LIN {X 0,Y 234.876,Z 433.115,A -85,B 0,C 180,E1 -19741.921,E2 -19741.921} C_VEL
LIN {X 0,Y 235.179,Z 429.868,A -85,B 0,C 180,E1 -19746.209,E2 -19746.209} C_VEL
LIN {X 0,Y 235.105,Z 427.906,A -85,B 0,C 180,E1 -19748.993,E2 -19748.993} C_VEL
LIN {X 0,Y 234.901,Z 426.222,A -85,B 0,C 180,E1 -19751.584,E2 -19751.584} C_VEL
LIN {X 0,Y 234.9,Z 426.223,A -85,B 0,C 180,E1 -19755.895,E2 -19755.895} C_VEL
LIN {X 0,Y 234.9,Z 426.226,A -85,B 0,C 180,E1 -19758.835,E2 -19758.835} C_VEL
LIN {X 0,Y 234.957,Z 426.217,A -85,B 0,C 180,E1 -19761.086,E2 -19761.086} C_VEL
LIN {X 0,Y 234.963,Z 426.216,A -85,B 0,C 180,E1 -19765.367,E2 -19765.367} C_VEL
LIN {X 0,Y 234.926,Z 426.22,A -85,B 0,C 180,E1 -19769.431,E2 -19769.431} C_VEL
LIN {X 0,Y 234.996,Z 426.211,A -85,B 0,C 180,E1 -19773.794,E2 -19773.794} C_VEL
LIN {X 0,Y 235.015,Z 426.21,A -85,B 0,C 180,E1 -19778.97,E2 -19778.97} C_VEL
LIN {X 0,Y 235.099,Z 426.198,A -85,B 0,C 180,E1 -19783.059,E2 -19783.059} C_VEL
LIN {X 0,Y 235.15,Z 426.194,A -85,B 0,C 180,E1 -19787.924,E2 -19787.924} C_VEL
LIN {X 0,Y 235.393,Z 426.161,A -85,B 0,C 180,E1 -19791.415,E2 -19791.415} C_VEL
LIN {X 0,Y 235.409,Z 426.16,A -85,B 0,C 180,E1 -19793.141,E2 -19793.141} C_VEL
LIN {X 0,Y 235.598,Z 426.138,A -85,B 0,C 180,E1 -19798.29,E2 -19798.29} C_VEL
LIN {X 0,Y 235.599,Z 426.139,A -85,B 0,C 180,E1 -19801.709,E2 -19801.709} C_VEL
LIN {X 0,Y 235.409,Z 426.161,A -85,B 0,C 180,E1 -19806.858,E2 -19806.858} C_VEL
LIN {X 0,Y 235.256,Z 426.178,A -85,B 0,C 180,E1 -19810.326,E2 -19810.326} C_VEL
LIN {X 0,Y 235.117,Z 426.198,A -85,B 0,C 180,E1 -19815.606,E2 -19815.606} C_VEL
LIN {X 0,Y 235.012,Z 426.212,A -85,B 0,C 180,E1 -19819.205,E2 -19819.205} C_VEL
LIN {X 0,Y 234.964,Z 426.216,A -85,B 0,C 180,E1 -19822.883,E2 -19822.883} C_VEL
LIN {X 0,Y 234.97,Z 426.215,A -85,B 0,C 180,E1 -19826.657,E2 -19826.657} C_VEL
LIN {X 0,Y 234.924,Z 426.222,A -85,B 0,C 180,E1 -19830.569,E2 -19830.569} C_VEL
LIN {X 0,Y 234.929,Z 426.22,A -85,B 0,C 180,E1 -19834.638,E2 -19834.638} C_VEL
LIN {X 0,Y 234.966,Z 426.376,A -85,B 0,C 180,E1 -19838.637,E2 -19838.637} C_VEL
LIN {X 0,Y 235.348,Z 428.729,A -85,B 0,C 180,E1 -19841.707,E2 -19841.707} C_VEL
LIN {X 0,Y 235.874,Z 431.984,A -85,B 0,C 180,E1 -19845.651,E2 -19845.651} C_VEL
LIN {X 0,Y 236.373,Z 435.044,A -85,B 0,C 180,E1 -19849.147,E2 -19849.147} C_VEL
LIN {X 0,Y 236.611,Z 436.635,A -85,B 0,C 180,E1 -19850.894,E2 -19850.894} C_VEL
LIN {X 0,Y 235.984,Z 437.599,A -85,B 0,C 180,E1 -19851.808,E2 -19851.808} C_VEL
LIN {X 0,Y 233.134,Z 439.375,A -85,B 0,C 180,E1 -19853.223,E2 -19853.223} C_VEL
LIN {X 0,Y 230.123,Z 441.18,A -85,B 0,C 180,E1 -19854.668,E2 -19854.668} C_VEL
LIN {X 0,Y 229.299,Z 442.206,A -85,B 0,C 180,E1 -19855.619,E2 -19855.619} C_VEL
LIN {X 0,Y 228.924,Z 443.785,A -85,B 0,C 180,E1 -19857.192,E2 -19857.192} C_VEL
LIN {X 0,Y 229.837,Z 447.058,A -85,B 0,C 180,E1 -19857.512,E2 -19857.512} C_VEL
LIN {X 0,Y 233.319,Z 459.076,A -85,B 0,C 180,E1 -19858.865,E2 -19858.865} C_VEL
LIN {X 0,Y 235.842,Z 471.592,A -85,B 0,C 180,E1 -19860.433,E2 -19860.433} C_VEL
LIN {X 0,Y 237.294,Z 482.933,A -85,B 0,C 180,E1 -19862.06,E2 -19862.06} C_VEL
LIN {X 0,Y 237.835,Z 494.199,A -85,B 0,C 180,E1 -19863.924,E2 -19863.924} C_VEL
LIN {X 0,Y 237.645,Z 500.432,A -85,B 0,C 180,E1 -19865.075,E2 -19865.075} C_VEL
LIN {X 0,Y 235.035,Z 510.888,A -85,B 0,C 180,E1 -19867.125,E2 -19867.125} C_VEL
LIN {X 0,Y 232.818,Z 519.781,A -85,B 0,C 180,E1 -19869.356,E2 -19869.356} C_VEL
LIN {X 0,Y 230.662,Z 527.628,A -85,B 0,C 180,E1 -19871.802,E2 -19871.802} C_VEL
LIN {X 0,Y 228.811,Z 534.295,A -85,B 0,C 180,E1 -19874.409,E2 -19874.409} C_VEL
LIN {X 0,Y 227.212,Z 540.397,A -85,B 0,C 180,E1 -19877.495,E2 -19877.495} C_VEL
LIN {X 0,Y 226.338,Z 544.368,A -85,B 0,C 180,E1 -19880.167,E2 -19880.167} C_VEL
LIN {X 0,Y 225.822,Z 547.305,A -85,B 0,C 180,E1 -19882.849,E2 -19882.849} C_VEL
LIN {X 0,Y 225.58,Z 549.275,A -85,B 0,C 180,E1 -19885.539,E2 -19885.539} C_VEL
LIN {X 0,Y 225.644,Z 550.313,A -85,B 0,C 180,E1 -19888.215,E2 -19888.215} C_VEL
LIN {X 0,Y 225.717,Z 550.528,A -85,B 0,C 180,E1 -19890,E2 -19890} C_VEL
LIN {X 0,Y 225.644,Z 550.303,A -85,B 0,C 180,E1 -19891.785,E2 -19891.785} C_VEL
LIN {X 0,Y 225.59,Z 549.231,A -85,B 0,C 180,E1 -19894.494,E2 -19894.494} C_VEL
LIN {X 0,Y 225.822,Z 547.272,A -85,B 0,C 180,E1 -19897.151,E2 -19897.151} C_VEL
LIN {X 0,Y 226.338,Z 544.321,A -85,B 0,C 180,E1 -19899.833,E2 -19899.833} C_VEL
LIN {X 0,Y 227.211,Z 540.331,A -85,B 0,C 180,E1 -19902.505,E2 -19902.505} C_VEL
LIN {X 0,Y 228.811,Z 534.203,A -85,B 0,C 180,E1 -19905.59,E2 -19905.59} C_VEL
LIN {X 0,Y 230.66,Z 527.515,A -85,B 0,C 180,E1 -19908.198,E2 -19908.198} C_VEL
LIN {X 0,Y 232.86,Z 519.542,A -85,B 0,C 180,E1 -19910.671,E2 -19910.671} C_VEL
LIN {X 0,Y 235.031,Z 510.713,A -85,B 0,C 180,E1 -19912.875,E2 -19912.875} C_VEL
LIN {X 0,Y 237.621,Z 500.209,A -85,B 0,C 180,E1 -19914.927,E2 -19914.927} C_VEL
LIN {X 0,Y 237.682,Z 491.057,A -85,B 0,C 180,E1 -19916.586,E2 -19916.586} C_VEL
LIN {X 0,Y 236.988,Z 480.028,A -85,B 0,C 180,E1 -19918.326,E2 -19918.326} C_VEL
LIN {X 0,Y 235.228,Z 468.348,A -85,B 0,C 180,E1 -19919.952,E2 -19919.952} C_VEL
LIN {X 0,Y 232.386,Z 455.412,A -85,B 0,C 180,E1 -19921.511,E2 -19921.511} C_VEL
LIN {X 0,Y 229.009,Z 444.333,A -85,B 0,C 180,E1 -19922.71,E2 -19922.71} C_VEL
LIN {X 0,Y 228.968,Z 443.753,A -85,B 0,C 180,E1 -19922.786,E2 -19922.786} C_VEL
LIN {X 0,Y 229.564,Z 440.977,A -85,B 0,C 180,E1 -19925.569,E2 -19925.569} C_VEL
LIN {X 0,Y 229.614,Z 437.882,A -85,B 0,C 180,E1 -19928.863,E2 -19928.863} C_VEL
LIN {X 0,Y 229.109,Z 434.593,A -85,B 0,C 180,E1 -19932.59,E2 -19932.59} C_VEL
LIN {X 0,Y 228.455,Z 430.668,A -85,B 0,C 180,E1 -19937.407,E2 -19937.407} C_VEL
LIN {X 0,Y 227.928,Z 427.099,A -85,B 0,C 180,E1 -19942.313,E2 -19942.313} C_VEL
LIN {X 0,Y 227.88,Z 427.104,A -85,B 0,C 180,E1 -19946.377,E2 -19946.377} C_VEL
LIN {X 0,Y 227.905,Z 427.099,A -85,B 0,C 180,E1 -19950.436,E2 -19950.436} C_VEL
LIN {X 0,Y 227.929,Z 427.094,A -85,B 0,C 180,E1 -19954.426,E2 -19954.426} C_VEL
LIN {X 0,Y 227.963,Z 427.091,A -85,B 0,C 180,E1 -19958.287,E2 -19958.287} C_VEL
LIN {X 0,Y 228.036,Z 427.082,A -85,B 0,C 180,E1 -19962.826,E2 -19962.826} C_VEL
LIN {X 0,Y 228.096,Z 427.072,A -85,B 0,C 180,E1 -19967.545,E2 -19967.545} C_VEL
LIN {X 0,Y 228.327,Z 427.043,A -85,B 0,C 180,E1 -19971.147,E2 -19971.147} C_VEL
LIN {X 0,Y 228.36,Z 427.036,A -85,B 0,C 180,E1 -19972.929,E2 -19972.929} C_VEL
LIN {X 0,Y 228.556,Z 427.016,A -85,B 0,C 180,E1 -19978.238,E2 -19978.238} C_VEL
LIN {X 0,Y 228.556,Z 427.015,A -85,B 0,C 180,E1 -19981.762,E2 -19981.762} C_VEL
LIN {X 0,Y 228.36,Z 427.038,A -85,B 0,C 180,E1 -19987.071,E2 -19987.071} C_VEL
LIN {X 0,Y 228.173,Z 427.061,A -85,B 0,C 180,E1 -19990.65,E2 -19990.65} C_VEL
LIN {X 0,Y 228.059,Z 427.077,A -85,B 0,C 180,E1 -19996.102,E2 -19996.102} C_VEL
LIN {X 0,Y 227.944,Z 427.087,A -85,B 0,C 180,E1 -19999.825,E2 -19999.825} C_VEL
LIN {X 0,Y 227.915,Z 427.096,A -85,B 0,C 180,E1 -20003.633,E2 -20003.633} C_VEL
LIN {X 0,Y 227.887,Z 427.099,A -85,B 0,C 180,E1 -20007.555,E2 -20007.555} C_VEL
LIN {X 0,Y 227.874,Z 427.101,A -85,B 0,C 180,E1 -20011.622,E2 -20011.622} C_VEL
LIN {X 0,Y 227.901,Z 427.096,A -85,B 0,C 180,E1 -20015.868,E2 -20015.868} C_VEL
LIN {X 0,Y 227.835,Z 427.104,A -85,B 0,C 180,E1 -20020.375,E2 -20020.375} C_VEL
LIN {X 0,Y 227.837,Z 427.106,A -85,B 0,C 180,E1 -20025.192,E2 -20025.192} C_VEL
LIN {X 0,Y 227.821,Z 427.109,A -85,B 0,C 180,E1 -20027.763,E2 -20027.763} C_VEL
LIN {X 0,Y 228.026,Z 428.595,A -85,B 0,C 180,E1 -20030.402,E2 -20030.402} C_VEL
LIN {X 0,Y 228.119,Z 431.17,A -85,B 0,C 180,E1 -20034.172,E2 -20034.172} C_VEL
LIN {X 0,Y 227.972,Z 433.391,A -85,B 0,C 180,E1 -20037.172,E2 -20037.172} C_VEL
LIN {X 0,Y 229.01,Z 436.551,A -85,B 0,C 180,E1 -20037.515,E2 -20037.515} C_VEL
LIN {X 0,Y 233.221,Z 448,A -85,B 0,C 180,E1 -20038.982,E2 -20038.982} C_VEL
LIN {X 0,Y 236.368,Z 459.105,A -85,B 0,C 180,E1 -20040.527,E2 -20040.527} C_VEL
LIN {X 0,Y 238.444,Z 469.825,A -85,B 0,C 180,E1 -20042.158,E2 -20042.158} C_VEL
LIN {X 0,Y 239.727,Z 480.037,A -85,B 0,C 180,E1 -20043.912,E2 -20043.912} C_VEL
LIN {X 0,Y 239.755,Z 482.646,A -85,B 0,C 180,E1 -20044.382,E2 -20044.382} C_VEL
LIN {X 0,Y 237.488,Z 493.091,A -85,B 0,C 180,E1 -20046.222,E2 -20046.222} C_VEL
LIN {X 0,Y 235.441,Z 501.875,A -85,B 0,C 180,E1 -20048.159,E2 -20048.159} C_VEL
LIN {X 0,Y 232.943,Z 510.862,A -85,B 0,C 180,E1 -20050.617,E2 -20050.617} C_VEL
LIN {X 0,Y 230.757,Z 518.268,A -85,B 0,C 180,E1 -20053.182,E2 -20053.182} C_VEL
LIN {X 0,Y 229.037,Z 524.207,A -85,B 0,C 180,E1 -20055.79,E2 -20055.79} C_VEL
LIN {X 0,Y 227.689,Z 528.899,A -85,B 0,C 180,E1 -20058.426,E2 -20058.426} C_VEL
LIN {X 0,Y 226.768,Z 532.486,A -85,B 0,C 180,E1 -20061.086,E2 -20061.086} C_VEL
LIN {X 0,Y 226.108,Z 535.319,A -85,B 0,C 180,E1 -20064.068,E2 -20064.068} C_VEL
LIN {X 0,Y 225.867,Z 536.717,A -85,B 0,C 180,E1 -20066.432,E2 -20066.432} C_VEL
LIN {X 0,Y 225.748,Z 537.552,A -85,B 0,C 180,E1 -20070,E2 -20070} C_VEL
LIN {X 0,Y 225.753,Z 537.359,A -85,B 0,C 180,E1 -20071.784,E2 -20071.784} C_VEL
LIN {X 0,Y 225.866,Z 536.773,A -85,B 0,C 180,E1 -20073.568,E2 -20073.568} C_VEL
LIN {X 0,Y 226.334,Z 534.45,A -85,B 0,C 180,E1 -20077.135,E2 -20077.135} C_VEL
LIN {X 0,Y 227.024,Z 531.583,A -85,B 0,C 180,E1 -20079.803,E2 -20079.803} C_VEL
LIN {X 0,Y 228.079,Z 527.693,A -85,B 0,C 180,E1 -20082.457,E2 -20082.457} C_VEL
LIN {X 0,Y 229.532,Z 522.672,A -85,B 0,C 180,E1 -20085.086,E2 -20085.086} C_VEL
LIN {X 0,Y 231.355,Z 516.347,A -85,B 0,C 180,E1 -20087.685,E2 -20087.685} C_VEL
LIN {X 0,Y 233.68,Z 508.429,A -85,B 0,C 180,E1 -20090.235,E2 -20090.235} C_VEL
LIN {X 0,Y 235.682,Z 500.566,A -85,B 0,C 180,E1 -20092.293,E2 -20092.293} C_VEL
LIN {X 0,Y 238.072,Z 490.511,A -85,B 0,C 180,E1 -20094.412,E2 -20094.412} C_VEL
LIN {X 0,Y 239.88,Z 482.103,A -85,B 0,C 180,E1 -20095.837,E2 -20095.837} C_VEL
LIN {X 0,Y 238.84,Z 471.948,A -85,B 0,C 180,E1 -20097.622,E2 -20097.622} C_VEL
LIN {X 0,Y 236.695,Z 460.288,A -85,B 0,C 180,E1 -20099.439,E2 -20099.439} C_VEL
LIN {X 0,Y 233.574,Z 448.999,A -85,B 0,C 180,E1 -20101.025,E2 -20101.025} C_VEL
LIN {X 0,Y 229.182,Z 436.839,A -85,B 0,C 180,E1 -20102.586,E2 -20102.586} C_VEL
LIN {X 0,Y 227.977,Z 433.327,A -85,B 0,C 180,E1 -20103.023,E2 -20103.023} C_VEL
LIN {X 0,Y 228.157,Z 430.599,A -85,B 0,C 180,E1 -20106.785,E2 -20106.785} C_VEL
LIN {X 0,Y 227.985,Z 428.215,A -85,B 0,C 180,E1 -20110.343,E2 -20110.343} C_VEL
LIN {X 0,Y 227.824,Z 427.103,A -85,B 0,C 180,E1 -20112.238,E2 -20112.238} C_VEL
LIN {X 0,Y 227.838,Z 427.104,A -85,B 0,C 180,E1 -20115.192,E2 -20115.192} C_VEL
LIN {X 0,Y 227.836,Z 427.103,A -85,B 0,C 180,E1 -20119.625,E2 -20119.625} C_VEL
LIN {X 0,Y 227.902,Z 427.095,A -85,B 0,C 180,E1 -20124.132,E2 -20124.132} C_VEL
LIN {X 0,Y 227.872,Z 427.101,A -85,B 0,C 180,E1 -20128.378,E2 -20128.378} C_VEL
LIN {X 0,Y 227.882,Z 427.1,A -85,B 0,C 180,E1 -20132.444,E2 -20132.444} C_VEL
LIN {X 0,Y 227.917,Z 427.096,A -85,B 0,C 180,E1 -20136.368,E2 -20136.368} C_VEL
LIN {X 0,Y 227.946,Z 427.091,A -85,B 0,C 180,E1 -20140.175,E2 -20140.175} C_VEL
LIN {X 0,Y 228.061,Z 427.077,A -85,B 0,C 180,E1 -20143.898,E2 -20143.898} C_VEL
LIN {X 0,Y 228.174,Z 427.062,A -85,B 0,C 180,E1 -20149.35,E2 -20149.35} C_VEL
LIN {X 0,Y 228.361,Z 427.038,A -85,B 0,C 180,E1 -20152.929,E2 -20152.929} C_VEL
LIN {X 0,Y 228.557,Z 427.015,A -85,B 0,C 180,E1 -20158.238,E2 -20158.238} C_VEL
LIN {X 0,Y 228.558,Z 427.016,A -85,B 0,C 180,E1 -20161.762,E2 -20161.762} C_VEL
LIN {X 0,Y 228.361,Z 427.039,A -85,B 0,C 180,E1 -20167.071,E2 -20167.071} C_VEL
LIN {X 0,Y 228.174,Z 427.06,A -85,B 0,C 180,E1 -20170.65,E2 -20170.65} C_VEL
LIN {X 0,Y 228.06,Z 427.077,A -85,B 0,C 180,E1 -20176.102,E2 -20176.102} C_VEL
LIN {X 0,Y 227.945,Z 427.091,A -85,B 0,C 180,E1 -20179.825,E2 -20179.825} C_VEL
LIN {X 0,Y 227.917,Z 427.095,A -85,B 0,C 180,E1 -20183.632,E2 -20183.632} C_VEL
LIN {X 0,Y 227.881,Z 427.098,A -85,B 0,C 180,E1 -20187.556,E2 -20187.556} C_VEL
LIN {X 0,Y 227.869,Z 427.093,A -85,B 0,C 180,E1 -20191.623,E2 -20191.623} C_VEL
LIN {X 0,Y 227.882,Z 427.098,A -85,B 0,C 180,E1 -20195.872,E2 -20195.872} C_VEL
LIN {X 0,Y 227.929,Z 427.222,A -85,B 0,C 180,E1 -20197.88,E2 -20197.88} C_VEL
LIN {X 0,Y 228.462,Z 430.743,A -85,B 0,C 180,E1 -20202.592,E2 -20202.592} C_VEL
LIN {X 0,Y 228.782,Z 432.699,A -85,B 0,C 180,E1 -20205.045,E2 -20205.045} C_VEL
LIN {X 0,Y 229.313,Z 435.857,A -85,B 0,C 180,E1 -20208.782,E2 -20208.782} C_VEL
LIN {X 0,Y 229.629,Z 438.973,A -85,B 0,C 180,E1 -20212.257,E2 -20212.257} C_VEL
LIN {X 0,Y 229.56,Z 441.027,A -85,B 0,C 180,E1 -20214.43,E2 -20214.43} C_VEL
LIN {X 0,Y 229.299,Z 442.206,A -85,B 0,C 180,E1 -20215.619,E2 -20215.619} C_VEL
LIN {X 0,Y 229.36,Z 443.899,A -85,B 0,C 180,E1 -20216.45,E2 -20216.45} C_VEL
LIN {X 0,Y 229.668,Z 446.642,A -85,B 0,C 180,E1 -20217.102,E2 -20217.102} C_VEL
LIN {X 0,Y 230.066,Z 451.856,A -85,B 0,C 180,E1 -20217.799,E2 -20217.799} C_VEL
LIN {X 0,Y 229.581,Z 462.151,A -85,B 0,C 180,E1 -20218.575,E2 -20218.575} C_VEL
LIN {X 0,Y 228.882,Z 468.288,A -85,B 0,C 180,E1 -20219.093,E2 -20219.093} C_VEL
LIN {X 0,Y 228.999,Z 470.221,A -85,B 0,C 180,E1 -20219.327,E2 -20219.327} C_VEL
LIN {X 0,Y 230.592,Z 481.763,A -85,B 0,C 180,E1 -20221.038,E2 -20221.038} C_VEL
LIN {X 0,Y 231.158,Z 492.673,A -85,B 0,C 180,E1 -20222.867,E2 -20222.867} C_VEL
LIN {X 0,Y 230.941,Z 501.408,A -85,B 0,C 180,E1 -20224.542,E2 -20224.542} C_VEL
LIN {X 0,Y 228.484,Z 510.686,A -85,B 0,C 180,E1 -20226.43,E2 -20226.43} C_VEL
LIN {X 0,Y 225.941,Z 520.317,A -85,B 0,C 180,E1 -20228.934,E2 -20228.934} C_VEL
LIN {X 0,Y 223.909,Z 527.425,A -85,B 0,C 180,E1 -20231.233,E2 -20231.233} C_VEL
LIN {X 0,Y 221.938,Z 534.091,A -85,B 0,C 180,E1 -20233.914,E2 -20233.914} C_VEL
LIN {X 0,Y 220.231,Z 540.193,A -85,B 0,C 180,E1 -20237.092,E2 -20237.092} C_VEL
LIN {X 0,Y 219.323,Z 544.164,A -85,B 0,C 180,E1 -20239.849,E2 -20239.849} C_VEL
LIN {X 0,Y 218.76,Z 547.101,A -85,B 0,C 180,E1 -20242.617,E2 -20242.617} C_VEL
LIN {X 0,Y 218.481,Z 549.232,A -85,B 0,C 180,E1 -20245.708,E2 -20245.708} C_VEL
LIN {X 0,Y 218.542,Z 550.109,A -85,B 0,C 180,E1 -20248.157,E2 -20248.157} C_VEL
LIN {X 0,Y 218.631,Z 550.325,A -85,B 0,C 180,E1 -20250,E2 -20250} C_VEL
LIN {X 0,Y 218.542,Z 550.099,A -85,B 0,C 180,E1 -20251.843,E2 -20251.843} C_VEL
LIN {X 0,Y 218.488,Z 549.205,A -85,B 0,C 180,E1 -20254.315,E2 -20254.315} C_VEL
LIN {X 0,Y 218.76,Z 547.067,A -85,B 0,C 180,E1 -20257.383,E2 -20257.383} C_VEL
LIN {X 0,Y 219.323,Z 544.115,A -85,B 0,C 180,E1 -20260.151,E2 -20260.151} C_VEL
LIN {X 0,Y 220.231,Z 540.124,A -85,B 0,C 180,E1 -20262.908,E2 -20262.908} C_VEL
LIN {X 0,Y 221.937,Z 533.996,A -85,B 0,C 180,E1 -20266.086,E2 -20266.086} C_VEL
LIN {X 0,Y 223.907,Z 527.308,A -85,B 0,C 180,E1 -20268.767,E2 -20268.767} C_VEL
LIN {X 0,Y 226.344,Z 518.762,A -85,B 0,C 180,E1 -20271.477,E2 -20271.477} C_VEL
LIN {X 0,Y 228.48,Z 510.505,A -85,B 0,C 180,E1 -20273.57,E2 -20273.57} C_VEL
LIN {X 0,Y 231.06,Z 499.997,A -85,B 0,C 180,E1 -20275.685,E2 -20275.685} C_VEL
LIN {X 0,Y 231.047,Z 489.297,A -85,B 0,C 180,E1 -20277.676,E2 -20277.676} C_VEL
LIN {X 0,Y 230.189,Z 478.595,A -85,B 0,C 180,E1 -20279.412,E2 -20279.412} C_VEL
LIN {X 0,Y 228.305,Z 466.709,A -85,B 0,C 180,E1 -20281.111,E2 -20281.111} C_VEL
LIN {X 0,Y 225.499,Z 454.685,A -85,B 0,C 180,E1 -20282.624,E2 -20282.624} C_VEL
LIN {X 0,Y 222.259,Z 444.269,A -85,B 0,C 180,E1 -20283.826,E2 -20283.826} C_VEL
LIN {X 0,Y 222.193,Z 443.529,A -85,B 0,C 180,E1 -20283.907,E2 -20283.907} C_VEL
LIN {X 0,Y 222.599,Z 439.832,A -85,B 0,C 180,E1 -20287.879,E2 -20287.879} C_VEL
LIN {X 0,Y 222.399,Z 437.38,A -85,B 0,C 180,E1 -20290.675,E2 -20290.675} C_VEL
LIN {X 0,Y 221.861,Z 434.498,A -85,B 0,C 180,E1 -20294.179,E2 -20294.179} C_VEL
LIN {X 0,Y 221.353,Z 431.385,A -85,B 0,C 180,E1 -20298.183,E2 -20298.183} C_VEL
LIN {X 0,Y 220.856,Z 427.981,A -85,B 0,C 180,E1 -20303.013,E2 -20303.013} C_VEL
LIN {X 0,Y 220.817,Z 427.983,A -85,B 0,C 180,E1 -20307.244,E2 -20307.244} C_VEL
LIN {X 0,Y 220.828,Z 427.978,A -85,B 0,C 180,E1 -20311.485,E2 -20311.485} C_VEL
LIN {X 0,Y 220.868,Z 427.972,A -85,B 0,C 180,E1 -20315.565,E2 -20315.565} C_VEL
LIN {X 0,Y 220.894,Z 427.97,A -85,B 0,C 180,E1 -20319.514,E2 -20319.514} C_VEL
LIN {X 0,Y 221.018,Z 427.954,A -85,B 0,C 180,E1 -20323.37,E2 -20323.37} C_VEL
LIN {X 0,Y 221.118,Z 427.941,A -85,B 0,C 180,E1 -20329.006,E2 -20329.006} C_VEL
LIN {X 0,Y 221.313,Z 427.915,A -85,B 0,C 180,E1 -20332.702,E2 -20332.702} C_VEL
LIN {X 0,Y 221.514,Z 427.892,A -85,B 0,C 180,E1 -20338.182,E2 -20338.182} C_VEL
LIN {X 0,Y 221.514,Z 427.893,A -85,B 0,C 180,E1 -20341.818,E2 -20341.818} C_VEL
LIN {X 0,Y 221.313,Z 427.916,A -85,B 0,C 180,E1 -20347.298,E2 -20347.298} C_VEL
LIN {X 0,Y 221.118,Z 427.939,A -85,B 0,C 180,E1 -20350.994,E2 -20350.994} C_VEL
LIN {X 0,Y 221.018,Z 427.953,A -85,B 0,C 180,E1 -20356.63,E2 -20356.63} C_VEL
LIN {X 0,Y 220.894,Z 427.968,A -85,B 0,C 180,E1 -20360.486,E2 -20360.486} C_VEL
LIN {X 0,Y 220.869,Z 427.971,A -85,B 0,C 180,E1 -20364.435,E2 -20364.435} C_VEL
LIN {X 0,Y 220.837,Z 427.975,A -85,B 0,C 180,E1 -20368.514,E2 -20368.514} C_VEL
LIN {X 0,Y 220.826,Z 427.976,A -85,B 0,C 180,E1 -20372.755,E2 -20372.755} C_VEL
LIN {X 0,Y 220.839,Z 427.977,A -85,B 0,C 180,E1 -20377.288,E2 -20377.288} C_VEL
LIN {X 0,Y 220.777,Z 427.985,A -85,B 0,C 180,E1 -20381.951,E2 -20381.951} C_VEL
LIN {X 0,Y 220.777,Z 427.985,A -85,B 0,C 180,E1 -20385.547,E2 -20385.547} C_VEL
LIN {X 0,Y 220.772,Z 427.986,A -85,B 0,C 180,E1 -20387.069,E2 -20387.069} C_VEL
LIN {X 0,Y 221.048,Z 429.859,A -85,B 0,C 180,E1 -20390.515,E2 -20390.515} C_VEL
LIN {X 0,Y 221.109,Z 431.393,A -85,B 0,C 180,E1 -20392.849,E2 -20392.849} C_VEL
LIN {X 0,Y 221.023,Z 433.72,A -85,B 0,C 180,E1 -20396.005,E2 -20396.005} C_VEL
LIN {X 0,Y 222.132,Z 436.853,A -85,B 0,C 180,E1 -20396.382,E2 -20396.382} C_VEL
LIN {X 0,Y 226.152,Z 447.303,A -85,B 0,C 180,E1 -20397.816,E2 -20397.816} C_VEL
LIN {X 0,Y 229.51,Z 458.684,A -85,B 0,C 180,E1 -20399.48,E2 -20399.48} C_VEL
LIN {X 0,Y 231.763,Z 470.005,A -85,B 0,C 180,E1 -20401.276,E2 -20401.276} C_VEL
LIN {X 0,Y 233.049,Z 480.257,A -85,B 0,C 180,E1 -20403.106,E2 -20403.106} C_VEL
LIN {X 0,Y 233.11,Z 484.141,A -85,B 0,C 180,E1 -20403.837,E2 -20403.837} C_VEL
LIN {X 0,Y 230.77,Z 494.355,A -85,B 0,C 180,E1 -20405.725,E2 -20405.725} C_VEL
LIN {X 0,Y 228.452,Z 503.743,A -85,B 0,C 180,E1 -20407.93,E2 -20407.93} C_VEL
LIN {X 0,Y 225.856,Z 512.416,A -85,B 0,C 180,E1 -20410.457,E2 -20410.457} C_VEL
LIN {X 0,Y 223.669,Z 519.583,A -85,B 0,C 180,E1 -20413.103,E2 -20413.103} C_VEL
LIN {X 0,Y 222.162,Z 524.412,A -85,B 0,C 180,E1 -20415.341,E2 -20415.341} C_VEL
LIN {X 0,Y 220.722,Z 529.104,A -85,B 0,C 180,E1 -20418.056,E2 -20418.056} C_VEL
LIN {X 0,Y 219.766,Z 532.69,A -85,B 0,C 180,E1 -20420.799,E2 -20420.799} C_VEL
LIN {X 0,Y 219,Z 535.748,A -85,B 0,C 180,E1 -20424.174,E2 -20424.174} C_VEL
LIN {X 0,Y 218.778,Z 536.921,A -85,B 0,C 180,E1 -20426.317,E2 -20426.317} C_VEL
LIN {X 0,Y 218.674,Z 537.529,A -85,B 0,C 180,E1 -20428.158,E2 -20428.158} C_VEL
LIN {X 0,Y 218.663,Z 537.756,A -85,B 0,C 180,E1 -20430,E2 -20430} C_VEL
LIN {X 0,Y 218.673,Z 537.563,A -85,B 0,C 180,E1 -20431.842,E2 -20431.842} C_VEL
LIN {X 0,Y 218.777,Z 536.977,A -85,B 0,C 180,E1 -20433.684,E2 -20433.684} C_VEL
LIN {X 0,Y 219.045,Z 535.757,A -85,B 0,C 180,E1 -20435.939,E2 -20435.939} C_VEL
LIN {X 0,Y 219.766,Z 532.84,A -85,B 0,C 180,E1 -20439.201,E2 -20439.201} C_VEL
LIN {X 0,Y 220.71,Z 529.31,A -85,B 0,C 180,E1 -20441.946,E2 -20441.946} C_VEL
LIN {X 0,Y 222.12,Z 524.673,A -85,B 0,C 180,E1 -20444.663,E2 -20444.663} C_VEL
LIN {X 0,Y 224.219,Z 517.684,A -85,B 0,C 180,E1 -20447.795,E2 -20447.795} C_VEL
LIN {X 0,Y 226.606,Z 510.101,A -85,B 0,C 180,E1 -20450.421,E2 -20450.421} C_VEL
LIN {X 0,Y 228.958,Z 501.382,A -85,B 0,C 180,E1 -20452.819,E2 -20452.819} C_VEL
LIN {X 0,Y 231.363,Z 491.777,A -85,B 0,C 180,E1 -20454.928,E2 -20454.928} C_VEL
LIN {X 0,Y 233.28,Z 483.589,A -85,B 0,C 180,E1 -20456.383,E2 -20456.383} C_VEL
LIN {X 0,Y 232.443,Z 474.156,A -85,B 0,C 180,E1 -20458.136,E2 -20458.136} C_VEL
LIN {X 0,Y 230.565,Z 463.118,A -85,B 0,C 180,E1 -20459.973,E2 -20459.973} C_VEL
LIN {X 0,Y 228.009,Z 453.076,A -85,B 0,C 180,E1 -20461.498,E2 -20461.498} C_VEL
LIN {X 0,Y 223.602,Z 440.285,A -85,B 0,C 180,E1 -20463.301,E2 -20463.301} C_VEL
LIN {X 0,Y 221.116,Z 434.19,A -85,B 0,C 180,E1 -20464.106,E2 -20464.106} C_VEL
LIN {X 0,Y 221.004,Z 433.54,A -85,B 0,C 180,E1 -20464.227,E2 -20464.227} C_VEL
LIN {X 0,Y 221.141,Z 431.337,A -85,B 0,C 180,E1 -20467.39,E2 -20467.39} C_VEL
LIN {X 0,Y 221.001,Z 429.484,A -85,B 0,C 180,E1 -20470.251,E2 -20470.251} C_VEL
LIN {X 0,Y 220.775,Z 427.981,A -85,B 0,C 180,E1 -20472.931,E2 -20472.931} C_VEL
LIN {X 0,Y 220.773,Z 427.985,A -85,B 0,C 180,E1 -20477.069,E2 -20477.069} C_VEL
LIN {X 0,Y 220.812,Z 427.981,A -85,B 0,C 180,E1 -20480.464,E2 -20480.464} C_VEL
LIN {X 0,Y 220.835,Z 427.978,A -85,B 0,C 180,E1 -20482.795,E2 -20482.795} C_VEL
LIN {X 0,Y 220.826,Z 427.975,A -85,B 0,C 180,E1 -20487.245,E2 -20487.245} C_VEL
LIN {X 0,Y 220.83,Z 427.976,A -85,B 0,C 180,E1 -20491.485,E2 -20491.485} C_VEL
LIN {X 0,Y 220.87,Z 427.97,A -85,B 0,C 180,E1 -20495.565,E2 -20495.565} C_VEL
LIN {X 0,Y 220.896,Z 427.968,A -85,B 0,C 180,E1 -20499.514,E2 -20499.514} C_VEL
LIN {X 0,Y 221.019,Z 427.952,A -85,B 0,C 180,E1 -20503.37,E2 -20503.37} C_VEL
LIN {X 0,Y 221.12,Z 427.94,A -85,B 0,C 180,E1 -20509.006,E2 -20509.006} C_VEL
LIN {X 0,Y 221.314,Z 427.916,A -85,B 0,C 180,E1 -20512.702,E2 -20512.702} C_VEL
LIN {X 0,Y 221.515,Z 427.893,A -85,B 0,C 180,E1 -20518.182,E2 -20518.182} C_VEL
LIN {X 0,Y 221.516,Z 427.892,A -85,B 0,C 180,E1 -20521.818,E2 -20521.818} C_VEL
LIN {X 0,Y 221.314,Z 427.918,A -85,B 0,C 180,E1 -20527.298,E2 -20527.298} C_VEL
LIN {X 0,Y 221.12,Z 427.94,A -85,B 0,C 180,E1 -20530.994,E2 -20530.994} C_VEL
LIN {X 0,Y 221.019,Z 427.953,A -85,B 0,C 180,E1 -20536.63,E2 -20536.63} C_VEL
LIN {X 0,Y 220.895,Z 427.968,A -85,B 0,C 180,E1 -20540.486,E2 -20540.486} C_VEL
LIN {X 0,Y 220.87,Z 427.971,A -85,B 0,C 180,E1 -20544.435,E2 -20544.435} C_VEL
LIN {X 0,Y 220.829,Z 427.973,A -85,B 0,C 180,E1 -20548.515,E2 -20548.515} C_VEL
LIN {X 0,Y 220.818,Z 427.963,A -85,B 0,C 180,E1 -20552.756,E2 -20552.756} C_VEL
LIN {X 0,Y 220.89,Z 428.16,A -85,B 0,C 180,E1 -20557.194,E2 -20557.194} C_VEL
LIN {X 0,Y 221.36,Z 431.471,A -85,B 0,C 180,E1 -20561.815,E2 -20561.815} C_VEL
LIN {X 0,Y 221.862,Z 434.559,A -85,B 0,C 180,E1 -20565.821,E2 -20565.821} C_VEL
LIN {X 0,Y 222.373,Z 437.454,A -85,B 0,C 180,E1 -20569.333,E2 -20569.333} C_VEL
LIN {X 0,Y 222.602,Z 439.883,A -85,B 0,C 180,E1 -20572.12,E2 -20572.12} C_VEL
LIN {X 0,Y 222.544,Z 441.825,A -85,B 0,C 180,E1 -20574.252,E2 -20574.252} C_VEL
LIN {X 0,Y 222.151,Z 443.548,A -85,B 0,C 180,E1 -20576.053,E2 -20576.053} C_VEL
LIN {X 0,Y 223.067,Z 446.896,A -85,B 0,C 180,E1 -20576.401,E2 -20576.401} C_VEL
LIN {X 0,Y 226.804,Z 459.479,A -85,B 0,C 180,E1 -20577.918,E2 -20577.918} C_VEL
LIN {X 0,Y 228.999,Z 470.221,A -85,B 0,C 180,E1 -20579.327,E2 -20579.327} C_VEL
LIN {X 0,Y 229.194,Z 475.519,A -85,B 0,C 180,E1 -20579.991,E2 -20579.991} C_VEL
LIN {X 0,Y 228.397,Z 480.869,A -85,B 0,C 180,E1 -20580.607,E2 -20580.607} C_VEL
LIN {X 0,Y 225.297,Z 492.988,A -85,B 0,C 180,E1 -20582.181,E2 -20582.181} C_VEL
LIN {X 0,Y 224.578,Z 497.835,A -85,B 0,C 180,E1 -20583.053,E2 -20583.053} C_VEL
LIN {X 0,Y 224.246,Z 502.333,A -85,B 0,C 180,E1 -20583.974,E2 -20583.974} C_VEL
LIN {X 0,Y 221.473,Z 512.28,A -85,B 0,C 180,E1 -20586.134,E2 -20586.134} C_VEL
LIN {X 0,Y 219.107,Z 520.782,A -85,B 0,C 180,E1 -20588.465,E2 -20588.465} C_VEL
LIN {X 0,Y 216.784,Z 528.459,A -85,B 0,C 180,E1 -20591.083,E2 -20591.083} C_VEL
LIN {X 0,Y 214.818,Z 534.883,A -85,B 0,C 180,E1 -20593.854,E2 -20593.854} C_VEL
LIN {X 0,Y 213.266,Z 539.988,A -85,B 0,C 180,E1 -20596.663,E2 -20596.663} C_VEL
LIN {X 0,Y 212.309,Z 543.96,A -85,B 0,C 180,E1 -20599.51,E2 -20599.51} C_VEL
LIN {X 0,Y 211.688,Z 546.896,A -85,B 0,C 180,E1 -20602.368,E2 -20602.368} C_VEL
LIN {X 0,Y 211.393,Z 549.152,A -85,B 0,C 180,E1 -20605.855,E2 -20605.855} C_VEL
LIN {X 0,Y 211.442,Z 549.905,A -85,B 0,C 180,E1 -20608.095,E2 -20608.095} C_VEL
LIN {X 0,Y 211.547,Z 550.121,A -85,B 0,C 180,E1 -20610,E2 -20610} C_VEL
LIN {X 0,Y 211.442,Z 549.894,A -85,B 0,C 180,E1 -20611.905,E2 -20611.905} C_VEL
LIN {X 0,Y 211.492,Z 548.271,A -85,B 0,C 180,E1 -20615.721,E2 -20615.721} C_VEL
LIN {X 0,Y 211.688,Z 546.861,A -85,B 0,C 180,E1 -20617.631,E2 -20617.631} C_VEL
LIN {X 0,Y 212.309,Z 543.909,A -85,B 0,C 180,E1 -20620.49,E2 -20620.49} C_VEL
LIN {X 0,Y 213.266,Z 539.917,A -85,B 0,C 180,E1 -20623.337,E2 -20623.337} C_VEL
LIN {X 0,Y 215.101,Z 533.79,A -85,B 0,C 180,E1 -20626.612,E2 -20626.612} C_VEL
LIN {X 0,Y 217.188,Z 527.102,A -85,B 0,C 180,E1 -20629.371,E2 -20629.371} C_VEL
LIN {X 0,Y 219.628,Z 518.869,A -85,B 0,C 180,E1 -20632.065,E2 -20632.065} C_VEL
LIN {X 0,Y 221.987,Z 510.298,A -85,B 0,C 180,E1 -20634.304,E2 -20634.304} C_VEL
LIN {X 0,Y 224.394,Z 500.966,A -85,B 0,C 180,E1 -20636.257,E2 -20636.257} C_VEL
LIN {X 0,Y 224.477,Z 490.217,A -85,B 0,C 180,E1 -20638.358,E2 -20638.358} C_VEL
LIN {X 0,Y 223.708,Z 479.579,A -85,B 0,C 180,E1 -20640.176,E2 -20640.176} C_VEL
LIN {X 0,Y 221.894,Z 467.664,A -85,B 0,C 180,E1 -20641.982,E2 -20641.982} C_VEL
LIN {X 0,Y 219.256,Z 456.069,A -85,B 0,C 180,E1 -20643.55,E2 -20643.55} C_VEL
LIN {X 0,Y 216.024,Z 445.968,A -85,B 0,C 180,E1 -20644.829,E2 -20644.829} C_VEL
LIN {X 0,Y 215.344,Z 443.298,A -85,B 0,C 180,E1 -20645.156,E2 -20645.156} C_VEL
LIN {X 0,Y 215.57,Z 440.315,A -85,B 0,C 180,E1 -20648.515,E2 -20648.515} C_VEL
LIN {X 0,Y 215.292,Z 437.961,A -85,B 0,C 180,E1 -20651.339,E2 -20651.339} C_VEL
LIN {X 0,Y 214.576,Z 433.889,A -85,B 0,C 180,E1 -20656.543,E2 -20656.543} C_VEL
LIN {X 0,Y 214.307,Z 432.098,A -85,B 0,C 180,E1 -20659.013,E2 -20659.013} C_VEL
LIN {X 0,Y 213.8,Z 428.86,A -85,B 0,C 180,E1 -20663.941,E2 -20663.941} C_VEL
LIN {X 0,Y 213.781,Z 428.859,A -85,B 0,C 180,E1 -20668.731,E2 -20668.731} C_VEL
LIN {X 0,Y 213.827,Z 428.851,A -85,B 0,C 180,E1 -20672.603,E2 -20672.603} C_VEL
LIN {X 0,Y 213.853,Z 428.848,A -85,B 0,C 180,E1 -20676.953,E2 -20676.953} C_VEL
LIN {X 0,Y 213.945,Z 428.837,A -85,B 0,C 180,E1 -20682.804,E2 -20682.804} C_VEL
LIN {X 0,Y 213.983,Z 428.832,A -85,B 0,C 180,E1 -20686.708,E2 -20686.708} C_VEL
LIN {X 0,Y 214.198,Z 428.804,A -85,B 0,C 180,E1 -20690.558,E2 -20690.558} C_VEL
LIN {X 0,Y 214.25,Z 428.796,A -85,B 0,C 180,E1 -20692.46,E2 -20692.46} C_VEL
LIN {X 0,Y 214.447,Z 428.772,A -85,B 0,C 180,E1 -20698.122,E2 -20698.122} C_VEL
LIN {X 0,Y 214.556,Z 428.759,A -85,B 0,C 180,E1 -20700,E2 -20700} C_VEL
LIN {X 0,Y 214.447,Z 428.773,A -85,B 0,C 180,E1 -20701.878,E2 -20701.878} C_VEL
LIN {X 0,Y 214.25,Z 428.797,A -85,B 0,C 180,E1 -20707.54,E2 -20707.54} C_VEL
LIN {X 0,Y 214.049,Z 428.82,A -85,B 0,C 180,E1 -20711.362,E2 -20711.362} C_VEL
LIN {X 0,Y 213.936,Z 428.836,A -85,B 0,C 180,E1 -20715.237,E2 -20715.237} C_VEL
LIN {X 0,Y 213.841,Z 428.843,A -85,B 0,C 180,E1 -20719.187,E2 -20719.187} C_VEL
LIN {X 0,Y 213.849,Z 428.846,A -85,B 0,C 180,E1 -20723.227,E2 -20723.227} C_VEL
LIN {X 0,Y 213.83,Z 428.849,A -85,B 0,C 180,E1 -20727.45,E2 -20727.45} C_VEL
LIN {X 0,Y 213.781,Z 428.856,A -85,B 0,C 180,E1 -20731.736,E2 -20731.736} C_VEL
LIN {X 0,Y 213.754,Z 428.858,A -85,B 0,C 180,E1 -20736.287,E2 -20736.287} C_VEL
LIN {X 0,Y 213.719,Z 428.864,A -85,B 0,C 180,E1 -20741.124,E2 -20741.124} C_VEL
LIN {X 0,Y 213.71,Z 428.864,A -85,B 0,C 180,E1 -20743.678,E2 -20743.678} C_VEL
LIN {X 0,Y 213.711,Z 428.867,A -85,B 0,C 180,E1 -20746.343,E2 -20746.343} C_VEL
LIN {X 0,Y 213.932,Z 430.195,A -85,B 0,C 180,E1 -20749.077,E2 -20749.077} C_VEL
LIN {X 0,Y 214.092,Z 431.99,A -85,B 0,C 180,E1 -20751.985,E2 -20751.985} C_VEL
LIN {X 0,Y 214.01,Z 433.796,A -85,B 0,C 180,E1 -20754.709,E2 -20754.709} C_VEL
LIN {X 0,Y 215.21,Z 437.146,A -85,B 0,C 180,E1 -20755.15,E2 -20755.15} C_VEL
LIN {X 0,Y 218.593,Z 445.359,A -85,B 0,C 180,E1 -20756.36,E2 -20756.36} C_VEL
LIN {X 0,Y 222.223,Z 456.62,A -85,B 0,C 180,E1 -20758.09,E2 -20758.09} C_VEL
LIN {X 0,Y 224.486,Z 466.327,A -85,B 0,C 180,E1 -20759.675,E2 -20759.675} C_VEL
LIN {X 0,Y 226.023,Z 477.029,A -85,B 0,C 180,E1 -20761.58,E2 -20761.58} C_VEL
LIN {X 0,Y 226.704,Z 484.351,A -85,B 0,C 180,E1 -20763.039,E2 -20763.039} C_VEL
LIN {X 0,Y 224.317,Z 494.558,A -85,B 0,C 180,E1 -20764.978,E2 -20764.978} C_VEL
LIN {X 0,Y 221.846,Z 504.097,A -85,B 0,C 180,E1 -20767.281,E2 -20767.281} C_VEL
LIN {X 0,Y 219.163,Z 512.623,A -85,B 0,C 180,E1 -20769.835,E2 -20769.835} C_VEL
LIN {X 0,Y 216.865,Z 519.789,A -85,B 0,C 180,E1 -20772.557,E2 -20772.557} C_VEL
LIN {X 0,Y 215.307,Z 524.618,A -85,B 0,C 180,E1 -20774.863,E2 -20774.863} C_VEL
LIN {X 0,Y 213.776,Z 529.31,A -85,B 0,C 180,E1 -20777.661,E2 -20777.661} C_VEL
LIN {X 0,Y 212.739,Z 532.896,A -85,B 0,C 180,E1 -20780.493,E2 -20780.493} C_VEL
LIN {X 0,Y 212.243,Z 534.747,A -85,B 0,C 180,E1 -20782.389,E2 -20782.389} C_VEL
LIN {X 0,Y 211.893,Z 536.137,A -85,B 0,C 180,E1 -20784.29,E2 -20784.29} C_VEL
LIN {X 0,Y 211.694,Z 537.125,A -85,B 0,C 180,E1 -20786.193,E2 -20786.193} C_VEL
LIN {X 0,Y 211.596,Z 537.732,A -85,B 0,C 180,E1 -20788.097,E2 -20788.097} C_VEL
LIN {X 0,Y 211.58,Z 537.96,A -85,B 0,C 180,E1 -20790,E2 -20790} C_VEL
LIN {X 0,Y 211.595,Z 537.766,A -85,B 0,C 180,E1 -20791.904,E2 -20791.904} C_VEL
LIN {X 0,Y 211.692,Z 537.181,A -85,B 0,C 180,E1 -20793.807,E2 -20793.807} C_VEL
LIN {X 0,Y 212.244,Z 534.857,A -85,B 0,C 180,E1 -20797.611,E2 -20797.611} C_VEL
LIN {X 0,Y 213.017,Z 531.99,A -85,B 0,C 180,E1 -20800.455,E2 -20800.455} C_VEL
LIN {X 0,Y 214.205,Z 528.099,A -85,B 0,C 180,E1 -20803.278,E2 -20803.278} C_VEL
LIN {X 0,Y 215.824,Z 523.078,A -85,B 0,C 180,E1 -20806.069,E2 -20806.069} C_VEL
LIN {X 0,Y 217.887,Z 516.751,A -85,B 0,C 180,E1 -20808.818,E2 -20808.818} C_VEL
LIN {X 0,Y 220.428,Z 508.831,A -85,B 0,C 180,E1 -20811.51,E2 -20811.51} C_VEL
LIN {X 0,Y 222.639,Z 500.77,A -85,B 0,C 180,E1 -20813.731,E2 -20813.731} C_VEL
LIN {X 0,Y 225.211,Z 490.913,A -85,B 0,C 180,E1 -20815.906,E2 -20815.906} C_VEL
LIN {X 0,Y 226.665,Z 485.076,A -85,B 0,C 180,E1 -20816.966,E2 -20816.966} C_VEL
LIN {X 0,Y 226.054,Z 476.407,A -85,B 0,C 180,E1 -20818.67,E2 -20818.67} C_VEL
LIN {X 0,Y 224.387,Z 465.585,A -85,B 0,C 180,E1 -20820.587,E2 -20820.587} C_VEL
LIN {X 0,Y 221.963,Z 455.663,A -85,B 0,C 180,E1 -20822.211,E2 -20822.211} C_VEL
LIN {X 0,Y 217.804,Z 443.237,A -85,B 0,C 180,E1 -20824.097,E2 -20824.097} C_VEL
LIN {X 0,Y 215.075,Z 436.861,A -85,B 0,C 180,E1 -20825.049,E2 -20825.049} C_VEL
LIN {X 0,Y 214.029,Z 433.772,A -85,B 0,C 180,E1 -20825.485,E2 -20825.485} C_VEL
LIN {X 0,Y 214.083,Z 431.733,A -85,B 0,C 180,E1 -20828.59,E2 -20828.59} C_VEL
LIN {X 0,Y 213.927,Z 430.208,A -85,B 0,C 180,E1 -20831.075,E2 -20831.075} C_VEL
LIN {X 0,Y 213.713,Z 428.861,A -85,B 0,C 180,E1 -20833.677,E2 -20833.677} C_VEL
LIN {X 0,Y 213.712,Z 428.864,A -85,B 0,C 180,E1 -20836.343,E2 -20836.343} C_VEL
LIN {X 0,Y 213.738,Z 428.859,A -85,B 0,C 180,E1 -20841.336,E2 -20841.336} C_VEL
LIN {X 0,Y 213.772,Z 428.858,A -85,B 0,C 180,E1 -20846.02,E2 -20846.02} C_VEL
LIN {X 0,Y 213.763,Z 428.855,A -85,B 0,C 180,E1 -20850.451,E2 -20850.451} C_VEL
LIN {X 0,Y 213.804,Z 428.849,A -85,B 0,C 180,E1 -20854.702,E2 -20854.702} C_VEL
LIN {X 0,Y 213.817,Z 428.851,A -85,B 0,C 180,E1 -20858.804,E2 -20858.804} C_VEL
LIN {X 0,Y 213.947,Z 428.834,A -85,B 0,C 180,E1 -20862.804,E2 -20862.804} C_VEL
LIN {X 0,Y 213.984,Z 428.83,A -85,B 0,C 180,E1 -20866.708,E2 -20866.708} C_VEL
LIN {X 0,Y 214.199,Z 428.801,A -85,B 0,C 180,E1 -20870.558,E2 -20870.558} C_VEL
LIN {X 0,Y 214.251,Z 428.797,A -85,B 0,C 180,E1 -20872.46,E2 -20872.46} C_VEL
LIN {X 0,Y 214.448,Z 428.773,A -85,B 0,C 180,E1 -20878.122,E2 -20878.122} C_VEL
LIN {X 0,Y 214.553,Z 428.759,A -85,B 0,C 180,E1 -20880,E2 -20880} C_VEL
LIN {X 0,Y 214.449,Z 428.772,A -85,B 0,C 180,E1 -20881.878,E2 -20881.878} C_VEL
LIN {X 0,Y 214.251,Z 428.798,A -85,B 0,C 180,E1 -20887.539,E2 -20887.539} C_VEL
LIN {X 0,Y 214.05,Z 428.821,A -85,B 0,C 180,E1 -20891.362,E2 -20891.362} C_VEL
LIN {X 0,Y 213.937,Z 428.837,A -85,B 0,C 180,E1 -20895.237,E2 -20895.237} C_VEL
LIN {X 0,Y 213.871,Z 428.846,A -85,B 0,C 180,E1 -20899.184,E2 -20899.184} C_VEL
LIN {X 0,Y 213.85,Z 428.848,A -85,B 0,C 180,E1 -20903.227,E2 -20903.227} C_VEL
LIN {X 0,Y 213.831,Z 428.848,A -85,B 0,C 180,E1 -20907.45,E2 -20907.45} C_VEL
LIN {X 0,Y 213.769,Z 428.845,A -85,B 0,C 180,E1 -20911.737,E2 -20911.737} C_VEL
LIN {X 0,Y 213.825,Z 428.975,A -85,B 0,C 180,E1 -20916.272,E2 -20916.272} C_VEL
LIN {X 0,Y 214.295,Z 432.219,A -85,B 0,C 180,E1 -20921.035,E2 -20921.035} C_VEL
LIN {X 0,Y 214.639,Z 434.331,A -85,B 0,C 180,E1 -20923.916,E2 -20923.916} C_VEL
LIN {X 0,Y 215.285,Z 438.021,A -85,B 0,C 180,E1 -20928.663,E2 -20928.663} C_VEL
LIN {X 0,Y 215.56,Z 440.576,A -85,B 0,C 180,E1 -20931.723,E2 -20931.723} C_VEL
LIN {X 0,Y 215.353,Z 443.352,A -85,B 0,C 180,E1 -20934.839,E2 -20934.839} C_VEL
LIN {X 0,Y 216.219,Z 446.474,A -85,B 0,C 180,E1 -20935.174,E2 -20935.174} C_VEL
LIN {X 0,Y 219.907,Z 458.452,A -85,B 0,C 180,E1 -20936.713,E2 -20936.713} C_VEL
LIN {X 0,Y 222.379,Z 470.167,A -85,B 0,C 180,E1 -20938.329,E2 -20938.329} C_VEL
LIN {X 0,Y 223.966,Z 481.592,A -85,B 0,C 180,E1 -20940.101,E2 -20940.101} C_VEL
LIN {X 0,Y 224.562,Z 492.463,A -85,B 0,C 180,E1 -20942.001,E2 -20942.001} C_VEL
LIN {X 0,Y 224.578,Z 497.835,A -85,B 0,C 180,E1 -20943.053,E2 -20943.053} C_VEL
LIN {X 0,Y 223.628,Z 501.039,A -85,B 0,C 180,E1 -20943.617,E2 -20943.617} C_VEL
LIN {X 0,Y 221.622,Z 504.099,A -85,B 0,C 180,E1 -20944.065,E2 -20944.065} C_VEL
LIN {X 0,Y 216.028,Z 510.725,A -85,B 0,C 180,E1 -20945.099,E2 -20945.099} C_VEL
LIN {X 0,Y 214.549,Z 513.555,A -85,B 0,C 180,E1 -20945.739,E2 -20945.739} C_VEL
LIN {X 0,Y 212.322,Z 521.172,A -85,B 0,C 180,E1 -20947.944,E2 -20947.944} C_VEL
LIN {X 0,Y 210.065,Z 528.256,A -85,B 0,C 180,E1 -20950.454,E2 -20950.454} C_VEL
LIN {X 0,Y 207.961,Z 534.679,A -85,B 0,C 180,E1 -20953.306,E2 -20953.306} C_VEL
LIN {X 0,Y 206.319,Z 539.784,A -85,B 0,C 180,E1 -20956.205,E2 -20956.205} C_VEL
LIN {X 0,Y 205.291,Z 543.756,A -85,B 0,C 180,E1 -20959.147,E2 -20959.147} C_VEL
LIN {X 0,Y 204.64,Z 546.693,A -85,B 0,C 180,E1 -20962.104,E2 -20962.104} C_VEL
LIN {X 0,Y 204.402,Z 548.09,A -85,B 0,C 180,E1 -20964.079,E2 -20964.079} C_VEL
LIN {X 0,Y 204.345,Z 549.701,A -85,B 0,C 180,E1 -20968.029,E2 -20968.029} C_VEL
LIN {X 0,Y 204.465,Z 549.917,A -85,B 0,C 180,E1 -20970,E2 -20970} C_VEL
LIN {X 0,Y 204.345,Z 549.69,A -85,B 0,C 180,E1 -20971.971,E2 -20971.971} C_VEL
LIN {X 0,Y 204.402,Z 548.066,A -85,B 0,C 180,E1 -20975.92,E2 -20975.92} C_VEL
LIN {X 0,Y 204.639,Z 546.656,A -85,B 0,C 180,E1 -20977.896,E2 -20977.896} C_VEL
LIN {X 0,Y 205.291,Z 543.703,A -85,B 0,C 180,E1 -20980.853,E2 -20980.853} C_VEL
LIN {X 0,Y 206.319,Z 539.711,A -85,B 0,C 180,E1 -20983.795,E2 -20983.795} C_VEL
LIN {X 0,Y 208.296,Z 533.584,A -85,B 0,C 180,E1 -20987.171,E2 -20987.171} C_VEL
LIN {X 0,Y 210.498,Z 526.896,A -85,B 0,C 180,E1 -20990.012,E2 -20990.012} C_VEL
LIN {X 0,Y 212.912,Z 519.015,A -85,B 0,C 180,E1 -20992.678,E2 -20992.678} C_VEL
LIN {X 0,Y 215.508,Z 510.09,A -85,B 0,C 180,E1 -20995.084,E2 -20995.084} C_VEL
LIN {X 0,Y 217.74,Z 501.904,A -85,B 0,C 180,E1 -20996.864,E2 -20996.864} C_VEL
LIN {X 0,Y 217.955,Z 491.965,A -85,B 0,C 180,E1 -20998.926,E2 -20998.926} C_VEL
LIN {X 0,Y 217.335,Z 481.145,A -85,B 0,C 180,E1 -21000.887,E2 -21000.887} C_VEL
LIN {X 0,Y 215.521,Z 468.694,A -85,B 0,C 180,E1 -21002.893,E2 -21002.893} C_VEL
LIN {X 0,Y 212.96,Z 457.072,A -85,B 0,C 180,E1 -21004.566,E2 -21004.566} C_VEL
LIN {X 0,Y 209.667,Z 446.845,A -85,B 0,C 180,E1 -21005.974,E2 -21005.974} C_VEL
LIN {X 0,Y 208.535,Z 443.724,A -85,B 0,C 180,E1 -21006.393,E2 -21006.393} C_VEL
LIN {X 0,Y 208.447,Z 443.086,A -85,B 0,C 180,E1 -21006.485,E2 -21006.485} C_VEL
LIN {X 0,Y 208.424,Z 440.271,A -85,B 0,C 180,E1 -21009.842,E2 -21009.842} C_VEL
LIN {X 0,Y 208.072,Z 438.198,A -85,B 0,C 180,E1 -21012.496,E2 -21012.496} C_VEL
LIN {X 0,Y 207.475,Z 434.582,A -85,B 0,C 180,E1 -21017.353,E2 -21017.353} C_VEL
LIN {X 0,Y 206.99,Z 431.235,A -85,B 0,C 180,E1 -21022.326,E2 -21022.326} C_VEL
LIN {X 0,Y 206.732,Z 429.74,A -85,B 0,C 180,E1 -21024.85,E2 -21024.85} C_VEL
LIN {X 0,Y 206.707,Z 429.738,A -85,B 0,C 180,E1 -21029.336,E2 -21029.336} C_VEL
LIN {X 0,Y 206.733,Z 429.732,A -85,B 0,C 180,E1 -21033.772,E2 -21033.772} C_VEL
LIN {X 0,Y 206.759,Z 429.731,A -85,B 0,C 180,E1 -21038.043,E2 -21038.043} C_VEL
LIN {X 0,Y 206.875,Z 429.717,A -85,B 0,C 180,E1 -21042.197,E2 -21042.197} C_VEL
LIN {X 0,Y 206.916,Z 429.711,A -85,B 0,C 180,E1 -21046.246,E2 -21046.246} C_VEL
LIN {X 0,Y 207.134,Z 429.684,A -85,B 0,C 180,E1 -21050.233,E2 -21050.233} C_VEL
LIN {X 0,Y 207.19,Z 429.677,A -85,B 0,C 180,E1 -21052.202,E2 -21052.202} C_VEL
LIN {X 0,Y 207.384,Z 429.652,A -85,B 0,C 180,E1 -21058.058,E2 -21058.058} C_VEL
LIN {X 0,Y 207.521,Z 429.635,A -85,B 0,C 180,E1 -21060,E2 -21060} C_VEL
LIN {X 0,Y 207.088,Z 429.689,A -85,B 0,C 180,E1 -21063.892,E2 -21063.892} C_VEL
LIN {X 0,Y 207.19,Z 429.677,A -85,B 0,C 180,E1 -21067.798,E2 -21067.798} C_VEL
LIN {X 0,Y 206.985,Z 429.702,A -85,B 0,C 180,E1 -21071.755,E2 -21071.755} C_VEL
LIN {X 0,Y 206.869,Z 429.716,A -85,B 0,C 180,E1 -21075.771,E2 -21075.771} C_VEL
LIN {X 0,Y 206.785,Z 429.722,A -85,B 0,C 180,E1 -21079.869,E2 -21079.869} C_VEL
LIN {X 0,Y 206.765,Z 429.73,A -85,B 0,C 180,E1 -21084.072,E2 -21084.072} C_VEL
LIN {X 0,Y 206.745,Z 429.731,A -85,B 0,C 180,E1 -21088.419,E2 -21088.419} C_VEL
LIN {X 0,Y 206.711,Z 429.734,A -85,B 0,C 180,E1 -21092.956,E2 -21092.956} C_VEL
LIN {X 0,Y 206.723,Z 429.735,A -85,B 0,C 180,E1 -21095.32,E2 -21095.32} C_VEL
LIN {X 0,Y 206.668,Z 429.741,A -85,B 0,C 180,E1 -21100.25,E2 -21100.25} C_VEL
LIN {X 0,Y 206.638,Z 429.746,A -85,B 0,C 180,E1 -21105.581,E2 -21105.581} C_VEL
LIN {X 0,Y 206.853,Z 431.038,A -85,B 0,C 180,E1 -21108.372,E2 -21108.372} C_VEL
LIN {X 0,Y 207.071,Z 433.414,A -85,B 0,C 180,E1 -21112.344,E2 -21112.344} C_VEL
LIN {X 0,Y 207.037,Z 434.098,A -85,B 0,C 180,E1 -21113.345,E2 -21113.345} C_VEL
LIN {X 0,Y 208.122,Z 437.169,A -85,B 0,C 180,E1 -21113.763,E2 -21113.763} C_VEL
LIN {X 0,Y 209.453,Z 439.932,A -85,B 0,C 180,E1 -21114.214,E2 -21114.214} C_VEL
LIN {X 0,Y 212.696,Z 447.883,A -85,B 0,C 180,E1 -21115.514,E2 -21115.514} C_VEL
LIN {X 0,Y 216.062,Z 458.846,A -85,B 0,C 180,E1 -21117.315,E2 -21117.315} C_VEL
LIN {X 0,Y 218.421,Z 469.712,A -85,B 0,C 180,E1 -21119.225,E2 -21119.225} C_VEL
LIN {X 0,Y 219.807,Z 480.697,A -85,B 0,C 180,E1 -21121.341,E2 -21121.341} C_VEL
LIN {X 0,Y 220.135,Z 485.835,A -85,B 0,C 180,E1 -21122.424,E2 -21122.424} C_VEL
LIN {X 0,Y 217.897,Z 494.766,A -85,B 0,C 180,E1 -21124.188,E2 -21124.188} C_VEL
LIN {X 0,Y 215.265,Z 504.448,A -85,B 0,C 180,E1 -21126.591,E2 -21126.591} C_VEL
LIN {X 0,Y 212.51,Z 512.83,A -85,B 0,C 180,E1 -21129.175,E2 -21129.175} C_VEL
LIN {X 0,Y 210.101,Z 519.995,A -85,B 0,C 180,E1 -21131.976,E2 -21131.976} C_VEL
LIN {X 0,Y 208.473,Z 524.823,A -85,B 0,C 180,E1 -21134.354,E2 -21134.354} C_VEL
LIN {X 0,Y 206.848,Z 529.515,A -85,B 0,C 180,E1 -21137.241,E2 -21137.241} C_VEL
LIN {X 0,Y 205.727,Z 533.101,A -85,B 0,C 180,E1 -21140.165,E2 -21140.165} C_VEL
LIN {X 0,Y 205.201,Z 534.952,A -85,B 0,C 180,E1 -21142.126,E2 -21142.126} C_VEL
LIN {X 0,Y 204.774,Z 536.542,A -85,B 0,C 180,E1 -21144.446,E2 -21144.446} C_VEL
LIN {X 0,Y 204.5,Z 537.937,A -85,B 0,C 180,E1 -21148.031,E2 -21148.031} C_VEL
LIN {X 0,Y 204.499,Z 538.163,A -85,B 0,C 180,E1 -21150,E2 -21150} C_VEL
LIN {X 0,Y 204.499,Z 537.97,A -85,B 0,C 180,E1 -21151.97,E2 -21151.97} C_VEL
LIN {X 0,Y 204.774,Z 536.619,A -85,B 0,C 180,E1 -21155.553,E2 -21155.553} C_VEL
LIN {X 0,Y 205.201,Z 535.061,A -85,B 0,C 180,E1 -21157.874,E2 -21157.874} C_VEL
LIN {X 0,Y 206.04,Z 532.193,A -85,B 0,C 180,E1 -21160.813,E2 -21160.813} C_VEL
LIN {X 0,Y 207.302,Z 528.302,A -85,B 0,C 180,E1 -21163.728,E2 -21163.728} C_VEL
LIN {X 0,Y 208.993,Z 523.281,A -85,B 0,C 180,E1 -21166.609,E2 -21166.609} C_VEL
LIN {X 0,Y 211.194,Z 516.952,A -85,B 0,C 180,E1 -21169.438,E2 -21169.438} C_VEL
LIN {X 0,Y 213.839,Z 509.033,A -85,B 0,C 180,E1 -21172.207,E2 -21172.207} C_VEL
LIN {X 0,Y 216.325,Z 500.356,A -85,B 0,C 180,E1 -21174.646,E2 -21174.646} C_VEL
LIN {X 0,Y 218.871,Z 491.112,A -85,B 0,C 180,E1 -21176.715,E2 -21176.715} C_VEL
LIN {X 0,Y 220.162,Z 485.282,A -85,B 0,C 180,E1 -21177.831,E2 -21177.831} C_VEL
LIN {X 0,Y 219.33,Z 475.563,A -85,B 0,C 180,E1 -21179.817,E2 -21179.817} C_VEL
LIN {X 0,Y 217.608,Z 465.145,A -85,B 0,C 180,E1 -21181.739,E2 -21181.739} C_VEL
LIN {X 0,Y 214.953,Z 454.78,A -85,B 0,C 180,E1 -21183.517,E2 -21183.517} C_VEL
LIN {X 0,Y 211.195,Z 443.919,A -85,B 0,C 180,E1 -21185.283,E2 -21185.283} C_VEL
LIN {X 0,Y 208.145,Z 437.154,A -85,B 0,C 180,E1 -21186.394,E2 -21186.394} C_VEL
LIN {X 0,Y 207.048,Z 434.027,A -85,B 0,C 180,E1 -21186.86,E2 -21186.86} C_VEL
LIN {X 0,Y 206.956,Z 431.992,A -85,B 0,C 180,E1 -21190.183,E2 -21190.183} C_VEL
LIN {X 0,Y 206.639,Z 429.743,A -85,B 0,C 180,E1 -21194.419,E2 -21194.419} C_VEL
LIN {X 0,Y 206.669,Z 429.74,A -85,B 0,C 180,E1 -21199.75,E2 -21199.75} C_VEL
LIN {X 0,Y 206.734,Z 429.733,A -85,B 0,C 180,E1 -21204.695,E2 -21204.695} C_VEL
LIN {X 0,Y 206.71,Z 429.735,A -85,B 0,C 180,E1 -21209.337,E2 -21209.337} C_VEL
LIN {X 0,Y 206.735,Z 429.73,A -85,B 0,C 180,E1 -21213.772,E2 -21213.772} C_VEL
LIN {X 0,Y 206.761,Z 429.73,A -85,B 0,C 180,E1 -21218.043,E2 -21218.043} C_VEL
LIN {X 0,Y 206.876,Z 429.715,A -85,B 0,C 180,E1 -21222.197,E2 -21222.197} C_VEL
LIN {X 0,Y 206.917,Z 429.712,A -85,B 0,C 180,E1 -21226.246,E2 -21226.246} C_VEL
LIN {X 0,Y 207.135,Z 429.682,A -85,B 0,C 180,E1 -21230.233,E2 -21230.233} C_VEL
LIN {X 0,Y 207.192,Z 429.678,A -85,B 0,C 180,E1 -21232.202,E2 -21232.202} C_VEL
LIN {X 0,Y 207.385,Z 429.654,A -85,B 0,C 180,E1 -21238.058,E2 -21238.058} C_VEL
LIN {X 0,Y 207.518,Z 429.635,A -85,B 0,C 180,E1 -21240,E2 -21240} C_VEL
LIN {X 0,Y 207.386,Z 429.652,A -85,B 0,C 180,E1 -21241.942,E2 -21241.942} C_VEL
LIN {X 0,Y 207.192,Z 429.676,A -85,B 0,C 180,E1 -21247.798,E2 -21247.798} C_VEL
LIN {X 0,Y 206.986,Z 429.704,A -85,B 0,C 180,E1 -21251.755,E2 -21251.755} C_VEL
LIN {X 0,Y 206.87,Z 429.716,A -85,B 0,C 180,E1 -21255.77,E2 -21255.77} C_VEL
LIN {X 0,Y 206.802,Z 429.724,A -85,B 0,C 180,E1 -21259.867,E2 -21259.867} C_VEL
LIN {X 0,Y 206.766,Z 429.728,A -85,B 0,C 180,E1 -21264.072,E2 -21264.072} C_VEL
LIN {X 0,Y 206.739,Z 429.728,A -85,B 0,C 180,E1 -21268.42,E2 -21268.42} C_VEL
LIN {X 0,Y 206.7,Z 429.72,A -85,B 0,C 180,E1 -21272.957,E2 -21272.957} C_VEL
LIN {X 0,Y 206.752,Z 429.826,A -85,B 0,C 180,E1 -21275.331,E2 -21275.331} C_VEL
LIN {X 0,Y 207.067,Z 431.949,A -85,B 0,C 180,E1 -21278.681,E2 -21278.681} C_VEL
LIN {X 0,Y 207.486,Z 434.66,A -85,B 0,C 180,E1 -21282.644,E2 -21282.644} C_VEL
LIN {X 0,Y 208.07,Z 438.255,A -85,B 0,C 180,E1 -21287.503,E2 -21287.503} C_VEL
LIN {X 0,Y 208.47,Z 440.883,A -85,B 0,C 180,E1 -21290.84,E2 -21290.84} C_VEL
LIN {X 0,Y 208.509,Z 443.156,A -85,B 0,C 180,E1 -21293.504,E2 -21293.504} C_VEL
LIN {X 0,Y 209.515,Z 446.428,A -85,B 0,C 180,E1 -21293.9,E2 -21293.9} C_VEL
LIN {X 0,Y 212.72,Z 456.34,A -85,B 0,C 180,E1 -21295.256,E2 -21295.256} C_VEL
LIN {X 0,Y 215.28,Z 466.832,A -85,B 0,C 180,E1 -21296.776,E2 -21296.776} C_VEL
LIN {X 0,Y 217.02,Z 478.375,A -85,B 0,C 180,E1 -21298.585,E2 -21298.585} C_VEL
LIN {X 0,Y 217.927,Z 489.403,A -85,B 0,C 180,E1 -21300.544,E2 -21300.544} C_VEL
LIN {X 0,Y 217.913,Z 499.811,A -85,B 0,C 180,E1 -21302.639,E2 -21302.639} C_VEL
LIN {X 0,Y 217.583,Z 503.204,A -85,B 0,C 180,E1 -21303.374,E2 -21303.374} C_VEL
LIN {X 0,Y 214.549,Z 513.555,A -85,B 0,C 180,E1 -21305.739,E2 -21305.739} C_VEL
LIN {X 0,Y 212.761,Z 517.642,A -85,B 0,C 180,E1 -21306.781,E2 -21306.781} C_VEL
LIN {X 0,Y 208.194,Z 523.835,A -85,B 0,C 180,E1 -21308.486,E2 -21308.486} C_VEL
LIN {X 0,Y 203.628,Z 529.385,A -85,B 0,C 180,E1 -21310.396,E2 -21310.396} C_VEL
LIN {X 0,Y 201.881,Z 532.466,A -85,B 0,C 180,E1 -21311.739,E2 -21311.739} C_VEL
LIN {X 0,Y 199.914,Z 537.99,A -85,B 0,C 180,E1 -21314.712,E2 -21314.712} C_VEL
LIN {X 0,Y 198.617,Z 542.327,A -85,B 0,C 180,E1 -21317.742,E2 -21317.742} C_VEL
LIN {X 0,Y 198.025,Z 544.626,A -85,B 0,C 180,E1 -21319.778,E2 -21319.778} C_VEL
LIN {X 0,Y 197.59,Z 546.489,A -85,B 0,C 180,E1 -21321.82,E2 -21321.82} C_VEL
LIN {X 0,Y 197.341,Z 547.887,A -85,B 0,C 180,E1 -21323.867,E2 -21323.867} C_VEL
LIN {X 0,Y 197.25,Z 549.498,A -85,B 0,C 180,E1 -21327.958,E2 -21327.958} C_VEL
LIN {X 0,Y 197.365,Z 549.713,A -85,B 0,C 180,E1 -21330,E2 -21330} C_VEL
LIN {X 0,Y 197.205,Z 549.005,A -85,B 0,C 180,E1 -21333.74,E2 -21333.74} C_VEL
LIN {X 0,Y 197.341,Z 547.861,A -85,B 0,C 180,E1 -21336.133,E2 -21336.133} C_VEL
LIN {X 0,Y 197.589,Z 546.451,A -85,B 0,C 180,E1 -21338.179,E2 -21338.179} C_VEL
LIN {X 0,Y 198.281,Z 543.497,A -85,B 0,C 180,E1 -21341.241,E2 -21341.241} C_VEL
LIN {X 0,Y 199.391,Z 539.505,A -85,B 0,C 180,E1 -21344.284,E2 -21344.284} C_VEL
LIN {X 0,Y 201.513,Z 533.378,A -85,B 0,C 180,E1 -21347.768,E2 -21347.768} C_VEL
LIN {X 0,Y 203.838,Z 526.69,A -85,B 0,C 180,E1 -21350.695,E2 -21350.695} C_VEL
LIN {X 0,Y 206.417,Z 518.531,A -85,B 0,C 180,E1 -21353.532,E2 -21353.532} C_VEL
LIN {X 0,Y 209.072,Z 509.882,A -85,B 0,C 180,E1 -21355.912,E2 -21355.912} C_VEL
LIN {X 0,Y 211.102,Z 502.77,A -85,B 0,C 180,E1 -21357.511,E2 -21357.511} C_VEL
LIN {X 0,Y 211.415,Z 491.745,A -85,B 0,C 180,E1 -21359.91,E2 -21359.91} C_VEL
LIN {X 0,Y 210.823,Z 481.458,A -85,B 0,C 180,E1 -21361.867,E2 -21361.867} C_VEL
LIN {X 0,Y 209.297,Z 470.135,A -85,B 0,C 180,E1 -21363.791,E2 -21363.791} C_VEL
LIN {X 0,Y 206.844,Z 458.905,A -85,B 0,C 180,E1 -21365.54,E2 -21365.54} C_VEL
LIN {X 0,Y 204.3,Z 450.48,A -85,B 0,C 180,E1 -21366.804,E2 -21366.804} C_VEL
LIN {X 0,Y 201.603,Z 443.532,A -85,B 0,C 180,E1 -21367.855,E2 -21367.855} C_VEL
LIN {X 0,Y 201.481,Z 442.804,A -85,B 0,C 180,E1 -21368.001,E2 -21368.001} C_VEL
LIN {X 0,Y 201.175,Z 440.013,A -85,B 0,C 180,E1 -21371.587,E2 -21371.587} C_VEL
LIN {X 0,Y 200.676,Z 437.142,A -85,B 0,C 180,E1 -21375.538,E2 -21375.538} C_VEL
LIN {X 0,Y 200.401,Z 435.289,A -85,B 0,C 180,E1 -21378.216,E2 -21378.216} C_VEL
LIN {X 0,Y 199.895,Z 432.029,A -85,B 0,C 180,E1 -21383.295,E2 -21383.295} C_VEL
LIN {X 0,Y 199.689,Z 430.616,A -85,B 0,C 180,E1 -21385.728,E2 -21385.728} C_VEL
LIN {X 0,Y 199.665,Z 430.616,A -85,B 0,C 180,E1 -21390.476,E2 -21390.476} C_VEL
LIN {X 0,Y 199.674,Z 430.613,A -85,B 0,C 180,E1 -21395.016,E2 -21395.016} C_VEL
LIN {X 0,Y 199.701,Z 430.61,A -85,B 0,C 180,E1 -21399.395,E2 -21399.395} C_VEL
LIN {X 0,Y 199.806,Z 430.597,A -85,B 0,C 180,E1 -21403.657,E2 -21403.657} C_VEL
LIN {X 0,Y 200.069,Z 430.563,A -85,B 0,C 180,E1 -21409.602,E2 -21409.602} C_VEL
LIN {X 0,Y 200.134,Z 430.556,A -85,B 0,C 180,E1 -21411.925,E2 -21411.925} C_VEL
LIN {X 0,Y 200.324,Z 430.531,A -85,B 0,C 180,E1 -21417.99,E2 -21417.99} C_VEL
LIN {X 0,Y 200.484,Z 430.511,A -85,B 0,C 180,E1 -21420,E2 -21420} C_VEL
LIN {X 0,Y 200.034,Z 430.569,A -85,B 0,C 180,E1 -21424.029,E2 -21424.029} C_VEL
LIN {X 0,Y 200.134,Z 430.555,A -85,B 0,C 180,E1 -21428.075,E2 -21428.075} C_VEL
LIN {X 0,Y 199.916,Z 430.583,A -85,B 0,C 180,E1 -21432.177,E2 -21432.177} C_VEL
LIN {X 0,Y 199.806,Z 430.596,A -85,B 0,C 180,E1 -21436.343,E2 -21436.343} C_VEL
LIN {X 0,Y 199.702,Z 430.608,A -85,B 0,C 180,E1 -21440.605,E2 -21440.605} C_VEL
LIN {X 0,Y 199.674,Z 430.612,A -85,B 0,C 180,E1 -21444.984,E2 -21444.984} C_VEL
LIN {X 0,Y 199.676,Z 430.612,A -85,B 0,C 180,E1 -21449.522,E2 -21449.522} C_VEL
LIN {X 0,Y 199.665,Z 430.612,A -85,B 0,C 180,E1 -21452.353,E2 -21452.353} C_VEL
LIN {X 0,Y 199.641,Z 430.616,A -85,B 0,C 180,E1 -21456.76,E2 -21456.76} C_VEL
LIN {X 0,Y 199.64,Z 430.617,A -85,B 0,C 180,E1 -21459.321,E2 -21459.321} C_VEL
LIN {X 0,Y 199.584,Z 430.627,A -85,B 0,C 180,E1 -21464.771,E2 -21464.771} C_VEL
LIN {X 0,Y 199.585,Z 430.625,A -85,B 0,C 180,E1 -21465.23,E2 -21465.23} C_VEL
LIN {X 0,Y 199.827,Z 432.133,A -85,B 0,C 180,E1 -21468.069,E2 -21468.069} C_VEL
LIN {X 0,Y 200.095,Z 434.399,A -85,B 0,C 180,E1 -21471.852,E2 -21471.852} C_VEL
LIN {X 0,Y 201.262,Z 437.576,A -85,B 0,C 180,E1 -21472.328,E2 -21472.328} C_VEL
LIN {X 0,Y 204.053,Z 443.446,A -85,B 0,C 180,E1 -21473.389,E2 -21473.389} C_VEL
LIN {X 0,Y 207.12,Z 451.334,A -85,B 0,C 180,E1 -21474.771,E2 -21474.771} C_VEL
LIN {X 0,Y 210.564,Z 463.475,A -85,B 0,C 180,E1 -21476.949,E2 -21476.949} C_VEL
LIN {X 0,Y 212.513,Z 474.343,A -85,B 0,C 180,E1 -21479.021,E2 -21479.021} C_VEL
LIN {X 0,Y 213.519,Z 484.789,A -85,B 0,C 180,E1 -21481.224,E2 -21481.224} C_VEL
LIN {X 0,Y 213.578,Z 487.225,A -85,B 0,C 180,E1 -21481.769,E2 -21481.769} C_VEL
LIN {X 0,Y 210.953,Z 496.927,A -85,B 0,C 180,E1 -21483.805,E2 -21483.805} C_VEL
LIN {X 0,Y 208.39,Z 505.751,A -85,B 0,C 180,E1 -21486.128,E2 -21486.128} C_VEL
LIN {X 0,Y 205.467,Z 514.362,A -85,B 0,C 180,E1 -21488.952,E2 -21488.952} C_VEL
LIN {X 0,Y 202.953,Z 521.227,A -85,B 0,C 180,E1 -21491.841,E2 -21491.841} C_VEL
LIN {X 0,Y 201.016,Z 526.719,A -85,B 0,C 180,E1 -21494.798,E2 -21494.798} C_VEL
LIN {X 0,Y 199.468,Z 531.028,A -85,B 0,C 180,E1 -21497.796,E2 -21497.796} C_VEL
LIN {X 0,Y 198.739,Z 533.306,A -85,B 0,C 180,E1 -21499.816,E2 -21499.816} C_VEL
LIN {X 0,Y 198.163,Z 535.157,A -85,B 0,C 180,E1 -21501.845,E2 -21501.845} C_VEL
LIN {X 0,Y 197.67,Z 536.926,A -85,B 0,C 180,E1 -21504.577,E2 -21504.577} C_VEL
LIN {X 0,Y 197.407,Z 538.141,A -85,B 0,C 180,E1 -21507.96,E2 -21507.96} C_VEL
LIN {X 0,Y 197.401,Z 538.367,A -85,B 0,C 180,E1 -21510,E2 -21510} C_VEL
LIN {X 0,Y 197.406,Z 538.174,A -85,B 0,C 180,E1 -21512.04,E2 -21512.04} C_VEL
LIN {X 0,Y 197.669,Z 537.002,A -85,B 0,C 180,E1 -21515.422,E2 -21515.422} C_VEL
LIN {X 0,Y 198.163,Z 535.264,A -85,B 0,C 180,E1 -21518.156,E2 -21518.156} C_VEL
LIN {X 0,Y 199.057,Z 532.397,A -85,B 0,C 180,E1 -21521.197,E2 -21521.197} C_VEL
LIN {X 0,Y 200.418,Z 528.505,A -85,B 0,C 180,E1 -21524.21,E2 -21524.21} C_VEL
LIN {X 0,Y 202.189,Z 523.484,A -85,B 0,C 180,E1 -21527.185,E2 -21527.185} C_VEL
LIN {X 0,Y 204.513,Z 517.154,A -85,B 0,C 180,E1 -21530.099,E2 -21530.099} C_VEL
LIN {X 0,Y 207.286,Z 509.234,A -85,B 0,C 180,E1 -21532.949,E2 -21532.949} C_VEL
LIN {X 0,Y 209.797,Z 500.842,A -85,B 0,C 180,E1 -21535.382,E2 -21535.382} C_VEL
LIN {X 0,Y 212.571,Z 491.312,A -85,B 0,C 180,E1 -21537.573,E2 -21537.573} C_VEL
LIN {X 0,Y 213.655,Z 486.705,A -85,B 0,C 180,E1 -21538.488,E2 -21538.488} C_VEL
LIN {X 0,Y 212.964,Z 477.508,A -85,B 0,C 180,E1 -21540.483,E2 -21540.483} C_VEL
LIN {X 0,Y 211.243,Z 466.298,A -85,B 0,C 180,E1 -21542.677,E2 -21542.677} C_VEL
LIN {X 0,Y 208.186,Z 454.648,A -85,B 0,C 180,E1 -21544.8,E2 -21544.8} C_VEL
LIN {X 0,Y 204.716,Z 444.935,A -85,B 0,C 180,E1 -21546.509,E2 -21546.509} C_VEL
LIN {X 0,Y 201.365,Z 437.694,A -85,B 0,C 180,E1 -21547.807,E2 -21547.807} C_VEL
LIN {X 0,Y 200.153,Z 434.748,A -85,B 0,C 180,E1 -21548.283,E2 -21548.283} C_VEL
LIN {X 0,Y 200.071,Z 434.26,A -85,B 0,C 180,E1 -21548.404,E2 -21548.404} C_VEL
LIN {X 0,Y 199.813,Z 431.978,A -85,B 0,C 180,E1 -21552.385,E2 -21552.385} C_VEL
LIN {X 0,Y 199.585,Z 430.623,A -85,B 0,C 180,E1 -21555.23,E2 -21555.23} C_VEL
LIN {X 0,Y 199.641,Z 430.618,A -85,B 0,C 180,E1 -21560.679,E2 -21560.679} C_VEL
LIN {X 0,Y 199.636,Z 430.618,A -85,B 0,C 180,E1 -21565.718,E2 -21565.718} C_VEL
LIN {X 0,Y 199.699,Z 430.609,A -85,B 0,C 180,E1 -21568.136,E2 -21568.136} C_VEL
LIN {X 0,Y 199.688,Z 430.61,A -85,B 0,C 180,E1 -21572.772,E2 -21572.772} C_VEL
LIN {X 0,Y 199.741,Z 430.603,A -85,B 0,C 180,E1 -21577.229,E2 -21577.229} C_VEL
LIN {X 0,Y 199.799,Z 430.598,A -85,B 0,C 180,E1 -21581.757,E2 -21581.757} C_VEL
LIN {X 0,Y 199.851,Z 430.589,A -85,B 0,C 180,E1 -21585.749,E2 -21585.749} C_VEL
LIN {X 0,Y 200.078,Z 430.564,A -85,B 0,C 180,E1 -21589.884,E2 -21589.884} C_VEL
LIN {X 0,Y 200.135,Z 430.555,A -85,B 0,C 180,E1 -21591.925,E2 -21591.925} C_VEL
LIN {X 0,Y 200.325,Z 430.533,A -85,B 0,C 180,E1 -21597.989,E2 -21597.989} C_VEL
LIN {X 0,Y 200.482,Z 430.511,A -85,B 0,C 180,E1 -21600,E2 -21600} C_VEL
LIN {X 0,Y 200.035,Z 430.569,A -85,B 0,C 180,E1 -21604.029,E2 -21604.029} C_VEL
LIN {X 0,Y 200.135,Z 430.554,A -85,B 0,C 180,E1 -21608.075,E2 -21608.075} C_VEL
LIN {X 0,Y 199.918,Z 430.582,A -85,B 0,C 180,E1 -21612.177,E2 -21612.177} C_VEL
LIN {X 0,Y 199.809,Z 430.596,A -85,B 0,C 180,E1 -21616.343,E2 -21616.343} C_VEL
LIN {X 0,Y 199.826,Z 430.593,A -85,B 0,C 180,E1 -21618.453,E2 -21618.453} C_VEL
LIN {X 0,Y 199.739,Z 430.604,A -85,B 0,C 180,E1 -21623.817,E2 -21623.817} C_VEL
LIN {X 0,Y 199.71,Z 430.603,A -85,B 0,C 180,E1 -21628.384,E2 -21628.384} C_VEL
LIN {X 0,Y 199.657,Z 430.597,A -85,B 0,C 180,E1 -21633.216,E2 -21633.216} C_VEL
LIN {X 0,Y 199.69,Z 430.645,A -85,B 0,C 180,E1 -21634.271,E2 -21634.271} C_VEL
LIN {X 0,Y 200.148,Z 433.801,A -85,B 0,C 180,E1 -21639.42,E2 -21639.42} C_VEL
LIN {X 0,Y 200.702,Z 437.196,A -85,B 0,C 180,E1 -21644.455,E2 -21644.455} C_VEL
LIN {X 0,Y 201.169,Z 440.084,A -85,B 0,C 180,E1 -21648.411,E2 -21648.411} C_VEL
LIN {X 0,Y 201.486,Z 442.855,A -85,B 0,C 180,E1 -21651.988,E2 -21651.988} C_VEL
LIN {X 0,Y 202.496,Z 446.016,A -85,B 0,C 180,E1 -21652.426,E2 -21652.426} C_VEL
LIN {X 0,Y 204.556,Z 451.017,A -85,B 0,C 180,E1 -21653.221,E2 -21653.221} C_VEL
LIN {X 0,Y 207.946,Z 463.068,A -85,B 0,C 180,E1 -21655.041,E2 -21655.041} C_VEL
LIN {X 0,Y 209.972,Z 474.072,A -85,B 0,C 180,E1 -21656.802,E2 -21656.802} C_VEL
LIN {X 0,Y 211.254,Z 486.199,A -85,B 0,C 180,E1 -21658.96,E2 -21658.96} C_VEL
LIN {X 0,Y 211.432,Z 496.097,A -85,B 0,C 180,E1 -21660.94,E2 -21660.94} C_VEL
LIN {X 0,Y 211.171,Z 503,A -85,B 0,C 180,E1 -21662.498,E2 -21662.498} C_VEL
LIN {X 0,Y 208.523,Z 511.875,A -85,B 0,C 180,E1 -21664.55,E2 -21664.55} C_VEL
LIN {X 0,Y 206.008,Z 520.043,A -85,B 0,C 180,E1 -21666.902,E2 -21666.902} C_VEL
LIN {X 0,Y 203.381,Z 528.054,A -85,B 0,C 180,E1 -21669.784,E2 -21669.784} C_VEL
LIN {X 0,Y 201.881,Z 532.466,A -85,B 0,C 180,E1 -21671.739,E2 -21671.739} C_VEL
LIN {X 0,Y 200.21,Z 535.337,A -85,B 0,C 180,E1 -21673.137,E2 -21673.137} C_VEL
LIN {X 0,Y 196.025,Z 539.498,A -85,B 0,C 180,E1 -21675.443,E2 -21675.443} C_VEL
LIN {X 0,Y 192.134,Z 542.919,A -85,B 0,C 180,E1 -21677.938,E2 -21677.938} C_VEL
LIN {X 0,Y 190.959,Z 544.596,A -85,B 0,C 180,E1 -21679.595,E2 -21679.595} C_VEL
LIN {X 0,Y 190.539,Z 546.284,A -85,B 0,C 180,E1 -21681.515,E2 -21681.515} C_VEL
LIN {X 0,Y 190.279,Z 547.683,A -85,B 0,C 180,E1 -21683.638,E2 -21683.638} C_VEL
LIN {X 0,Y 190.157,Z 549.294,A -85,B 0,C 180,E1 -21687.882,E2 -21687.882} C_VEL
LIN {X 0,Y 190.268,Z 549.509,A -85,B 0,C 180,E1 -21690,E2 -21690} C_VEL
LIN {X 0,Y 190.122,Z 548.925,A -85,B 0,C 180,E1 -21693.554,E2 -21693.554} C_VEL
LIN {X 0,Y 190.279,Z 547.656,A -85,B 0,C 180,E1 -21696.362,E2 -21696.362} C_VEL
LIN {X 0,Y 190.539,Z 546.246,A -85,B 0,C 180,E1 -21698.484,E2 -21698.484} C_VEL
LIN {X 0,Y 191.293,Z 543.291,A -85,B 0,C 180,E1 -21701.658,E2 -21701.658} C_VEL
LIN {X 0,Y 192.479,Z 539.298,A -85,B 0,C 180,E1 -21704.808,E2 -21704.808} C_VEL
LIN {X 0,Y 194.75,Z 533.172,A -85,B 0,C 180,E1 -21708.407,E2 -21708.407} C_VEL
LIN {X 0,Y 197.203,Z 526.484,A -85,B 0,C 180,E1 -21711.425,E2 -21711.425} C_VEL
LIN {X 0,Y 199.929,Z 518.185,A -85,B 0,C 180,E1 -21714.395,E2 -21714.395} C_VEL
LIN {X 0,Y 202.704,Z 509.675,A -85,B 0,C 180,E1 -21716.79,E2 -21716.79} C_VEL
LIN {X 0,Y 204.502,Z 503.634,A -85,B 0,C 180,E1 -21718.199,E2 -21718.199} C_VEL
LIN {X 0,Y 204.93,Z 493.052,A -85,B 0,C 180,E1 -21720.631,E2 -21720.631} C_VEL
LIN {X 0,Y 204.49,Z 483.148,A -85,B 0,C 180,E1 -21722.639,E2 -21722.639} C_VEL
LIN {X 0,Y 203.168,Z 471.89,A -85,B 0,C 180,E1 -21724.686,E2 -21724.686} C_VEL
LIN {X 0,Y 200.988,Z 461.235,A -85,B 0,C 180,E1 -21726.473,E2 -21726.473} C_VEL
LIN {X 0,Y 198.494,Z 453.012,A -85,B 0,C 180,E1 -21727.828,E2 -21727.828} C_VEL
LIN {X 0,Y 196.018,Z 446.727,A -85,B 0,C 180,E1 -21728.897,E2 -21728.897} C_VEL
LIN {X 0,Y 194.579,Z 443.563,A -85,B 0,C 180,E1 -21729.462,E2 -21729.462} C_VEL
LIN {X 0,Y 194.394,Z 442.583,A -85,B 0,C 180,E1 -21729.599,E2 -21729.599} C_VEL
LIN {X 0,Y 193.937,Z 439.735,A -85,B 0,C 180,E1 -21733.55,E2 -21733.55} C_VEL
LIN {X 0,Y 193.583,Z 437.675,A -85,B 0,C 180,E1 -21736.56,E2 -21736.56} C_VEL
LIN {X 0,Y 193.047,Z 434.349,A -85,B 0,C 180,E1 -21741.764,E2 -21741.764} C_VEL
LIN {X 0,Y 192.641,Z 431.615,A -85,B 0,C 180,E1 -21746.51,E2 -21746.51} C_VEL
LIN {X 0,Y 192.661,Z 431.487,A -85,B 0,C 180,E1 -21751.691,E2 -21751.691} C_VEL
LIN {X 0,Y 192.707,Z 431.482,A -85,B 0,C 180,E1 -21756.349,E2 -21756.349} C_VEL
LIN {X 0,Y 192.733,Z 431.478,A -85,B 0,C 180,E1 -21761.457,E2 -21761.457} C_VEL
LIN {X 0,Y 192.774,Z 431.473,A -85,B 0,C 180,E1 -21765.215,E2 -21765.215} C_VEL
LIN {X 0,Y 193.021,Z 431.441,A -85,B 0,C 180,E1 -21769.511,E2 -21769.511} C_VEL
LIN {X 0,Y 193.006,Z 431.437,A -85,B 0,C 180,E1 -21773.729,E2 -21773.729} C_VEL
LIN {X 0,Y 193.266,Z 431.41,A -85,B 0,C 180,E1 -21777.916,E2 -21777.916} C_VEL
LIN {X 0,Y 193.448,Z 431.388,A -85,B 0,C 180,E1 -21780,E2 -21780} C_VEL
LIN {X 0,Y 192.981,Z 431.448,A -85,B 0,C 180,E1 -21784.177,E2 -21784.177} C_VEL
LIN {X 0,Y 193.081,Z 431.433,A -85,B 0,C 180,E1 -21788.372,E2 -21788.372} C_VEL
LIN {X 0,Y 192.855,Z 431.461,A -85,B 0,C 180,E1 -21792.63,E2 -21792.63} C_VEL
LIN {X 0,Y 192.759,Z 431.474,A -85,B 0,C 180,E1 -21796.959,E2 -21796.959} C_VEL
LIN {X 0,Y 192.638,Z 431.489,A -85,B 0,C 180,E1 -21801.397,E2 -21801.397} C_VEL
LIN {X 0,Y 192.666,Z 431.485,A -85,B 0,C 180,E1 -21804.225,E2 -21804.225} C_VEL
LIN {X 0,Y 192.651,Z 431.486,A -85,B 0,C 180,E1 -21808.892,E2 -21808.892} C_VEL
LIN {X 0,Y 192.602,Z 431.493,A -85,B 0,C 180,E1 -21813.186,E2 -21813.186} C_VEL
LIN {X 0,Y 192.611,Z 431.492,A -85,B 0,C 180,E1 -21816.608,E2 -21816.608} C_VEL
LIN {X 0,Y 192.525,Z 431.504,A -85,B 0,C 180,E1 -21821.078,E2 -21821.078} C_VEL
LIN {X 0,Y 192.496,Z 431.506,A -85,B 0,C 180,E1 -21823.923,E2 -21823.923} C_VEL
LIN {X 0,Y 192.703,Z 432.754,A -85,B 0,C 180,E1 -21826.838,E2 -21826.838} C_VEL
LIN {X 0,Y 192.985,Z 434.537,A -85,B 0,C 180,E1 -21830.151,E2 -21830.151} C_VEL
LIN {X 0,Y 194.242,Z 437.815,A -85,B 0,C 180,E1 -21830.709,E2 -21830.709} C_VEL
LIN {X 0,Y 195.502,Z 439.96,A -85,B 0,C 180,E1 -21831.17,E2 -21831.17} C_VEL
LIN {X 0,Y 199.97,Z 450.307,A -85,B 0,C 180,E1 -21833.173,E2 -21833.173} C_VEL
LIN {X 0,Y 203.185,Z 460.699,A -85,B 0,C 180,E1 -21835.141,E2 -21835.141} C_VEL
LIN {X 0,Y 205.294,Z 470.094,A -85,B 0,C 180,E1 -21837.005,E2 -21837.005} C_VEL
LIN {X 0,Y 206.541,Z 479.689,A -85,B 0,C 180,E1 -21839.016,E2 -21839.016} C_VEL
LIN {X 0,Y 207.024,Z 488.602,A -85,B 0,C 180,E1 -21841.069,E2 -21841.069} C_VEL
LIN {X 0,Y 204.068,Z 499.076,A -85,B 0,C 180,E1 -21843.403,E2 -21843.403} C_VEL
LIN {X 0,Y 201.34,Z 507.552,A -85,B 0,C 180,E1 -21845.786,E2 -21845.786} C_VEL
LIN {X 0,Y 198.405,Z 515.794,A -85,B 0,C 180,E1 -21848.711,E2 -21848.711} C_VEL
LIN {X 0,Y 196.211,Z 521.433,A -85,B 0,C 180,E1 -21851.194,E2 -21851.194} C_VEL
LIN {X 0,Y 194.172,Z 526.924,A -85,B 0,C 180,E1 -21854.249,E2 -21854.249} C_VEL
LIN {X 0,Y 192.519,Z 531.234,A -85,B 0,C 180,E1 -21857.348,E2 -21857.348} C_VEL
LIN {X 0,Y 191.746,Z 533.511,A -85,B 0,C 180,E1 -21859.44,E2 -21859.44} C_VEL
LIN {X 0,Y 191.126,Z 535.362,A -85,B 0,C 180,E1 -21861.542,E2 -21861.542} C_VEL
LIN {X 0,Y 190.568,Z 537.307,A -85,B 0,C 180,E1 -21864.711,E2 -21864.711} C_VEL
LIN {X 0,Y 190.317,Z 538.345,A -85,B 0,C 180,E1 -21867.884,E2 -21867.884} C_VEL
LIN {X 0,Y 190.306,Z 538.571,A -85,B 0,C 180,E1 -21870,E2 -21870} C_VEL
LIN {X 0,Y 190.316,Z 538.377,A -85,B 0,C 180,E1 -21872.117,E2 -21872.117} C_VEL
LIN {X 0,Y 190.577,Z 537.366,A -85,B 0,C 180,E1 -21875.316,E2 -21875.316} C_VEL
LIN {X 0,Y 191.126,Z 535.468,A -85,B 0,C 180,E1 -21878.458,E2 -21878.458} C_VEL
LIN {X 0,Y 192.099,Z 532.6,A -85,B 0,C 180,E1 -21881.609,E2 -21881.609} C_VEL
LIN {X 0,Y 193.537,Z 528.708,A -85,B 0,C 180,E1 -21884.726,E2 -21884.726} C_VEL
LIN {X 0,Y 195.413,Z 523.686,A -85,B 0,C 180,E1 -21887.801,E2 -21887.801} C_VEL
LIN {X 0,Y 197.855,Z 517.356,A -85,B 0,C 180,E1 -21890.807,E2 -21890.807} C_VEL
LIN {X 0,Y 200.761,Z 509.436,A -85,B 0,C 180,E1 -21893.74,E2 -21893.74} C_VEL
LIN {X 0,Y 203.319,Z 501.27,A -85,B 0,C 180,E1 -21896.181,E2 -21896.181} C_VEL
LIN {X 0,Y 206.311,Z 491.512,A -85,B 0,C 180,E1 -21898.484,E2 -21898.484} C_VEL
LIN {X 0,Y 207.14,Z 488.074,A -85,B 0,C 180,E1 -21899.191,E2 -21899.191} C_VEL
LIN {X 0,Y 206.509,Z 478.624,A -85,B 0,C 180,E1 -21901.359,E2 -21901.359} C_VEL
LIN {X 0,Y 205.18,Z 469.056,A -85,B 0,C 180,E1 -21903.349,E2 -21903.349} C_VEL
LIN {X 0,Y 202.657,Z 458.579,A -85,B 0,C 180,E1 -21905.416,E2 -21905.416} C_VEL
LIN {X 0,Y 199.513,Z 449.034,A -85,B 0,C 180,E1 -21907.228,E2 -21907.228} C_VEL
LIN {X 0,Y 194.951,Z 438.781,A -85,B 0,C 180,E1 -21909.221,E2 -21909.221} C_VEL
LIN {X 0,Y 193.225,Z 435.617,A -85,B 0,C 180,E1 -21909.881,E2 -21909.881} C_VEL
LIN {X 0,Y 192.958,Z 434.499,A -85,B 0,C 180,E1 -21910.104,E2 -21910.104} C_VEL
LIN {X 0,Y 192.675,Z 432.48,A -85,B 0,C 180,E1 -21913.872,E2 -21913.872} C_VEL
LIN {X 0,Y 192.518,Z 431.504,A -85,B 0,C 180,E1 -21916.083,E2 -21916.083} C_VEL
LIN {X 0,Y 192.543,Z 431.5,A -85,B 0,C 180,E1 -21920.043,E2 -21920.043} C_VEL
LIN {X 0,Y 192.6,Z 431.492,A -85,B 0,C 180,E1 -21924.279,E2 -21924.279} C_VEL
LIN {X 0,Y 192.602,Z 431.493,A -85,B 0,C 180,E1 -21929.279,E2 -21929.279} C_VEL
LIN {X 0,Y 192.663,Z 431.485,A -85,B 0,C 180,E1 -21931.691,E2 -21931.691} C_VEL
LIN {X 0,Y 192.709,Z 431.482,A -85,B 0,C 180,E1 -21936.349,E2 -21936.349} C_VEL
LIN {X 0,Y 192.735,Z 431.477,A -85,B 0,C 180,E1 -21941.457,E2 -21941.457} C_VEL
LIN {X 0,Y 192.775,Z 431.47,A -85,B 0,C 180,E1 -21945.214,E2 -21945.214} C_VEL
LIN {X 0,Y 193.023,Z 431.441,A -85,B 0,C 180,E1 -21949.511,E2 -21949.511} C_VEL
LIN {X 0,Y 193.007,Z 431.442,A -85,B 0,C 180,E1 -21953.728,E2 -21953.728} C_VEL
LIN {X 0,Y 193.267,Z 431.412,A -85,B 0,C 180,E1 -21957.916,E2 -21957.916} C_VEL
LIN {X 0,Y 193.446,Z 431.388,A -85,B 0,C 180,E1 -21960,E2 -21960} C_VEL
LIN {X 0,Y 192.982,Z 431.447,A -85,B 0,C 180,E1 -21964.177,E2 -21964.177} C_VEL
LIN {X 0,Y 193.082,Z 431.433,A -85,B 0,C 180,E1 -21968.372,E2 -21968.372} C_VEL
LIN {X 0,Y 192.856,Z 431.461,A -85,B 0,C 180,E1 -21972.63,E2 -21972.63} C_VEL
LIN {X 0,Y 192.784,Z 431.471,A -85,B 0,C 180,E1 -21978.586,E2 -21978.586} C_VEL
LIN {X 0,Y 192.667,Z 431.484,A -85,B 0,C 180,E1 -21984.225,E2 -21984.225} C_VEL
LIN {X 0,Y 192.646,Z 431.483,A -85,B 0,C 180,E1 -21988.889,E2 -21988.889} C_VEL
LIN {X 0,Y 192.621,Z 431.497,A -85,B 0,C 180,E1 -21993.182,E2 -21993.182} C_VEL
LIN {X 0,Y 193.05,Z 434.416,A -85,B 0,C 180,E1 -21998.235,E2 -21998.235} C_VEL
LIN {X 0,Y 193.607,Z 437.845,A -85,B 0,C 180,E1 -22003.607,E2 -22003.607} C_VEL
LIN {X 0,Y 194.109,Z 440.874,A -85,B 0,C 180,E1 -22007.946,E2 -22007.946} C_VEL
LIN {X 0,Y 194.379,Z 442.651,A -85,B 0,C 180,E1 -22010.355,E2 -22010.355} C_VEL
LIN {X 0,Y 195.501,Z 445.89,A -85,B 0,C 180,E1 -22010.84,E2 -22010.84} C_VEL
LIN {X 0,Y 196.67,Z 448.176,A -85,B 0,C 180,E1 -22011.278,E2 -22011.278} C_VEL
LIN {X 0,Y 199.29,Z 455.012,A -85,B 0,C 180,E1 -22012.445,E2 -22012.445} C_VEL
LIN {X 0,Y 202.2,Z 466.234,A -85,B 0,C 180,E1 -22014.293,E2 -22014.293} C_VEL
LIN {X 0,Y 203.891,Z 476.786,A -85,B 0,C 180,E1 -22016.113,E2 -22016.113} C_VEL
LIN {X 0,Y 204.89,Z 488.282,A -85,B 0,C 180,E1 -22018.324,E2 -22018.324} C_VEL
LIN {X 0,Y 204.838,Z 498.649,A -85,B 0,C 180,E1 -22020.554,E2 -22020.554} C_VEL
LIN {X 0,Y 204.307,Z 504.945,A -85,B 0,C 180,E1 -22022.05,E2 -22022.05} C_VEL
LIN {X 0,Y 201.528,Z 513.46,A -85,B 0,C 180,E1 -22024.156,E2 -22024.156} C_VEL
LIN {X 0,Y 198.528,Z 522.701,A -85,B 0,C 180,E1 -22027.082,E2 -22027.082} C_VEL
LIN {X 0,Y 195.838,Z 530.127,A -85,B 0,C 180,E1 -22030.066,E2 -22030.066} C_VEL
LIN {X 0,Y 193.672,Z 536.094,A -85,B 0,C 180,E1 -22033.124,E2 -22033.124} C_VEL
LIN {X 0,Y 192.05,Z 540.812,A -85,B 0,C 180,E1 -22036.239,E2 -22036.239} C_VEL
LIN {X 0,Y 190.959,Z 544.596,A -85,B 0,C 180,E1 -22039.595,E2 -22039.595} C_VEL
LIN {X 0,Y 189.899,Z 546.112,A -85,B 0,C 180,E1 -22041.293,E2 -22041.293} C_VEL
LIN {X 0,Y 186.655,Z 547.885,A -85,B 0,C 180,E1 -22044.095,E2 -22044.095} C_VEL
LIN {X 0,Y 184.136,Z 548.801,A -85,B 0,C 180,E1 -22046.419,E2 -22046.419} C_VEL
LIN {X 0,Y 183.13,Z 549.179,A -85,B 0,C 180,E1 -22048.244,E2 -22048.244} C_VEL
LIN {X 0,Y 183.077,Z 549.194,A -85,B 0,C 180,E1 -22048.864,E2 -22048.864} C_VEL
LIN {X 0,Y 183.173,Z 549.305,A -85,B 0,C 180,E1 -22050,E2 -22050} C_VEL
LIN {X 0,Y 183.032,Z 548.832,A -85,B 0,C 180,E1 -22053.301,E2 -22053.301} C_VEL
LIN {X 0,Y 183.211,Z 547.452,A -85,B 0,C 180,E1 -22056.608,E2 -22056.608} C_VEL
LIN {X 0,Y 183.508,Z 546.041,A -85,B 0,C 180,E1 -22058.812,E2 -22058.812} C_VEL
LIN {X 0,Y 184.325,Z 543.086,A -85,B 0,C 180,E1 -22062.105,E2 -22062.105} C_VEL
LIN {X 0,Y 185.586,Z 539.092,A -85,B 0,C 180,E1 -22065.372,E2 -22065.372} C_VEL
LIN {X 0,Y 188.009,Z 532.966,A -85,B 0,C 180,E1 -22069.092,E2 -22069.092} C_VEL
LIN {X 0,Y 190.542,Z 526.409,A -85,B 0,C 180,E1 -22072.153,E2 -22072.153} C_VEL
LIN {X 0,Y 193.448,Z 517.977,A -85,B 0,C 180,E1 -22075.269,E2 -22075.269} C_VEL
LIN {X 0,Y 196.388,Z 509.468,A -85,B 0,C 180,E1 -22077.724,E2 -22077.724} C_VEL
LIN {X 0,Y 197.932,Z 504.499,A -85,B 0,C 180,E1 -22078.933,E2 -22078.933} C_VEL
LIN {X 0,Y 198.482,Z 494.007,A -85,B 0,C 180,E1 -22081.471,E2 -22081.471} C_VEL
LIN {X 0,Y 198.121,Z 483.804,A -85,B 0,C 180,E1 -22083.659,E2 -22083.659} C_VEL
LIN {X 0,Y 196.915,Z 472.665,A -85,B 0,C 180,E1 -22085.798,E2 -22085.798} C_VEL
LIN {X 0,Y 194.528,Z 460.993,A -85,B 0,C 180,E1 -22087.893,E2 -22087.893} C_VEL
LIN {X 0,Y 191.329,Z 451.486,A -85,B 0,C 180,E1 -22089.629,E2 -22089.629} C_VEL
LIN {X 0,Y 189.039,Z 446.709,A -85,B 0,C 180,E1 -22090.605,E2 -22090.605} C_VEL
LIN {X 0,Y 187.37,Z 443.35,A -85,B 0,C 180,E1 -22091.296,E2 -22091.296} C_VEL
LIN {X 0,Y 187.157,Z 442.37,A -85,B 0,C 180,E1 -22091.415,E2 -22091.415} C_VEL
LIN {X 0,Y 186.642,Z 439.483,A -85,B 0,C 180,E1 -22095.679,E2 -22095.679} C_VEL
LIN {X 0,Y 186.233,Z 436.709,A -85,B 0,C 180,E1 -22100.093,E2 -22100.093} C_VEL
LIN {X 0,Y 185.814,Z 433.64,A -85,B 0,C 180,E1 -22105.435,E2 -22105.435} C_VEL
LIN {X 0,Y 185.544,Z 432.376,A -85,B 0,C 180,E1 -22107.975,E2 -22107.975} C_VEL
LIN {X 0,Y 185.581,Z 432.37,A -85,B 0,C 180,E1 -22110.577,E2 -22110.577} C_VEL
LIN {X 0,Y 185.589,Z 432.367,A -85,B 0,C 180,E1 -22115.383,E2 -22115.383} C_VEL
LIN {X 0,Y 185.676,Z 432.358,A -85,B 0,C 180,E1 -22121.133,E2 -22121.133} C_VEL
LIN {X 0,Y 185.726,Z 432.351,A -85,B 0,C 180,E1 -22124.64,E2 -22124.64} C_VEL
LIN {X 0,Y 185.944,Z 432.323,A -85,B 0,C 180,E1 -22129.328,E2 -22129.328} C_VEL
LIN {X 0,Y 185.97,Z 432.314,A -85,B 0,C 180,E1 -22133.49,E2 -22133.49} C_VEL
LIN {X 0,Y 186.21,Z 432.289,A -85,B 0,C 180,E1 -22137.837,E2 -22137.837} C_VEL
LIN {X 0,Y 186.411,Z 432.264,A -85,B 0,C 180,E1 -22140,E2 -22140} C_VEL
LIN {X 0,Y 185.929,Z 432.325,A -85,B 0,C 180,E1 -22144.336,E2 -22144.336} C_VEL
LIN {X 0,Y 186.031,Z 432.312,A -85,B 0,C 180,E1 -22148.692,E2 -22148.692} C_VEL
LIN {X 0,Y 185.767,Z 432.344,A -85,B 0,C 180,E1 -22153.12,E2 -22153.12} C_VEL
LIN {X 0,Y 185.692,Z 432.355,A -85,B 0,C 180,E1 -22157.625,E2 -22157.625} C_VEL
LIN {X 0,Y 185.598,Z 432.365,A -85,B 0,C 180,E1 -22162.251,E2 -22162.251} C_VEL
LIN {X 0,Y 185.564,Z 432.369,A -85,B 0,C 180,E1 -22167.032,E2 -22167.032} C_VEL
LIN {X 0,Y 185.58,Z 432.368,A -85,B 0,C 180,E1 -22169.493,E2 -22169.493} C_VEL
LIN {X 0,Y 185.52,Z 432.374,A -85,B 0,C 180,E1 -22174.628,E2 -22174.628} C_VEL
LIN {X 0,Y 185.545,Z 432.373,A -85,B 0,C 180,E1 -22177.304,E2 -22177.304} C_VEL
LIN {X 0,Y 185.487,Z 432.38,A -85,B 0,C 180,E1 -22180.73,E2 -22180.73} C_VEL
LIN {X 0,Y 185.497,Z 432.65,A -85,B 0,C 180,E1 -22183.957,E2 -22183.957} C_VEL
LIN {X 0,Y 185.822,Z 434.769,A -85,B 0,C 180,E1 -22188.264,E2 -22188.264} C_VEL
LIN {X 0,Y 187.086,Z 437.952,A -85,B 0,C 180,E1 -22188.88,E2 -22188.88} C_VEL
LIN {X 0,Y 188.623,Z 440.425,A -85,B 0,C 180,E1 -22189.483,E2 -22189.483} C_VEL
LIN {X 0,Y 192.047,Z 447.601,A -85,B 0,C 180,E1 -22191.047,E2 -22191.047} C_VEL
LIN {X 0,Y 195.76,Z 457.645,A -85,B 0,C 180,E1 -22193.138,E2 -22193.138} C_VEL
LIN {X 0,Y 198.566,Z 469.037,A -85,B 0,C 180,E1 -22195.508,E2 -22195.508} C_VEL
LIN {X 0,Y 199.934,Z 478.283,A -85,B 0,C 180,E1 -22197.527,E2 -22197.527} C_VEL
LIN {X 0,Y 200.596,Z 488.818,A -85,B 0,C 180,E1 -22200.049,E2 -22200.049} C_VEL
LIN {X 0,Y 199.557,Z 493.268,A -85,B 0,C 180,E1 -22201.037,E2 -22201.037} C_VEL
LIN {X 0,Y 196.589,Z 502.81,A -85,B 0,C 180,E1 -22203.441,E2 -22203.441} C_VEL
LIN {X 0,Y 193.856,Z 510.715,A -85,B 0,C 180,E1 -22205.93,E2 -22205.93} C_VEL
LIN {X 0,Y 190.829,Z 518.393,A -85,B 0,C 180,E1 -22208.956,E2 -22208.956} C_VEL
LIN {X 0,Y 188.747,Z 523.635,A -85,B 0,C 180,E1 -22211.549,E2 -22211.549} C_VEL
LIN {X 0,Y 186.725,Z 528.715,A -85,B 0,C 180,E1 -22214.724,E2 -22214.724} C_VEL
LIN {X 0,Y 185.135,Z 532.659,A -85,B 0,C 180,E1 -22217.949,E2 -22217.949} C_VEL
LIN {X 0,Y 184.115,Z 535.567,A -85,B 0,C 180,E1 -22221.218,E2 -22221.218} C_VEL
LIN {X 0,Y 183.458,Z 537.685,A -85,B 0,C 180,E1 -22224.89,E2 -22224.89} C_VEL
LIN {X 0,Y 183.229,Z 538.549,A -85,B 0,C 180,E1 -22227.802,E2 -22227.802} C_VEL
LIN {X 0,Y 183.212,Z 538.775,A -85,B 0,C 180,E1 -22230,E2 -22230} C_VEL
LIN {X 0,Y 183.228,Z 538.581,A -85,B 0,C 180,E1 -22232.198,E2 -22232.198} C_VEL
LIN {X 0,Y 183.459,Z 537.737,A -85,B 0,C 180,E1 -22235.113,E2 -22235.113} C_VEL
LIN {X 0,Y 184.116,Z 535.671,A -85,B 0,C 180,E1 -22238.783,E2 -22238.783} C_VEL
LIN {X 0,Y 185.131,Z 532.804,A -85,B 0,C 180,E1 -22242.052,E2 -22242.052} C_VEL
LIN {X 0,Y 186.658,Z 528.911,A -85,B 0,C 180,E1 -22245.282,E2 -22245.282} C_VEL
LIN {X 0,Y 188.641,Z 523.89,A -85,B 0,C 180,E1 -22248.462,E2 -22248.462} C_VEL
LIN {X 0,Y 191.237,Z 517.558,A -85,B 0,C 180,E1 -22251.562,E2 -22251.562} C_VEL
LIN {X 0,Y 194.275,Z 509.638,A -85,B 0,C 180,E1 -22254.584,E2 -22254.584} C_VEL
LIN {X 0,Y 196.889,Z 501.745,A -85,B 0,C 180,E1 -22257.016,E2 -22257.016} C_VEL
LIN {X 0,Y 200.105,Z 491.713,A -85,B 0,C 180,E1 -22259.453,E2 -22259.453} C_VEL
LIN {X 0,Y 200.675,Z 489.444,A -85,B 0,C 180,E1 -22259.938,E2 -22259.938} C_VEL
LIN {X 0,Y 200.026,Z 478.762,A -85,B 0,C 180,E1 -22262.514,E2 -22262.514} C_VEL
LIN {X 0,Y 198.771,Z 469.959,A -85,B 0,C 180,E1 -22264.452,E2 -22264.452} C_VEL
LIN {X 0,Y 196.053,Z 458.556,A -85,B 0,C 180,E1 -22266.836,E2 -22266.836} C_VEL
LIN {X 0,Y 192.595,Z 448.97,A -85,B 0,C 180,E1 -22268.842,E2 -22268.842} C_VEL
LIN {X 0,Y 189.622,Z 442.458,A -85,B 0,C 180,E1 -22270.25,E2 -22270.25} C_VEL
LIN {X 0,Y 187.687,Z 438.835,A -85,B 0,C 180,E1 -22271.071,E2 -22271.071} C_VEL
LIN {X 0,Y 186.083,Z 435.838,A -85,B 0,C 180,E1 -22271.746,E2 -22271.746} C_VEL
LIN {X 0,Y 185.826,Z 434.758,A -85,B 0,C 180,E1 -22271.946,E2 -22271.946} C_VEL
LIN {X 0,Y 185.54,Z 432.741,A -85,B 0,C 180,E1 -22276.03,E2 -22276.03} C_VEL
LIN {X 0,Y 185.481,Z 432.381,A -85,B 0,C 180,E1 -22276.997,E2 -22276.997} C_VEL
LIN {X 0,Y 185.492,Z 432.378,A -85,B 0,C 180,E1 -22279.901,E2 -22279.901} C_VEL
LIN {X 0,Y 185.546,Z 432.374,A -85,B 0,C 180,E1 -22282.696,E2 -22282.696} C_VEL
LIN {X 0,Y 185.543,Z 432.371,A -85,B 0,C 180,E1 -22287.975,E2 -22287.975} C_VEL
LIN {X 0,Y 185.583,Z 432.364,A -85,B 0,C 180,E1 -22290.577,E2 -22290.577} C_VEL
LIN {X 0,Y 185.59,Z 432.365,A -85,B 0,C 180,E1 -22295.383,E2 -22295.383} C_VEL
LIN {X 0,Y 185.61,Z 432.364,A -85,B 0,C 180,E1 -22300.075,E2 -22300.075} C_VEL
LIN {X 0,Y 185.727,Z 432.348,A -85,B 0,C 180,E1 -22304.64,E2 -22304.64} C_VEL
LIN {X 0,Y 185.945,Z 432.322,A -85,B 0,C 180,E1 -22309.328,E2 -22309.328} C_VEL
LIN {X 0,Y 185.972,Z 432.319,A -85,B 0,C 180,E1 -22313.49,E2 -22313.49} C_VEL
LIN {X 0,Y 186.211,Z 432.29,A -85,B 0,C 180,E1 -22317.837,E2 -22317.837} C_VEL
LIN {X 0,Y 186.41,Z 432.264,A -85,B 0,C 180,E1 -22320,E2 -22320} C_VEL
LIN {X 0,Y 185.93,Z 432.325,A -85,B 0,C 180,E1 -22324.336,E2 -22324.336} C_VEL
LIN {X 0,Y 186.032,Z 432.311,A -85,B 0,C 180,E1 -22328.691,E2 -22328.691} C_VEL
LIN {X 0,Y 185.768,Z 432.344,A -85,B 0,C 180,E1 -22333.12,E2 -22333.12} C_VEL
LIN {X 0,Y 185.719,Z 432.351,A -85,B 0,C 180,E1 -22337.622,E2 -22337.622} C_VEL
LIN {X 0,Y 185.603,Z 432.364,A -85,B 0,C 180,E1 -22342.251,E2 -22342.251} C_VEL
LIN {X 0,Y 185.563,Z 432.372,A -85,B 0,C 180,E1 -22347.032,E2 -22347.032} C_VEL
LIN {X 0,Y 185.579,Z 432.366,A -85,B 0,C 180,E1 -22349.493,E2 -22349.493} C_VEL
LIN {X 0,Y 185.547,Z 432.373,A -85,B 0,C 180,E1 -22352.024,E2 -22352.024} C_VEL
LIN {X 0,Y 185.992,Z 435.173,A -85,B 0,C 180,E1 -22357.199,E2 -22357.199} C_VEL
LIN {X 0,Y 186.346,Z 437.461,A -85,B 0,C 180,E1 -22361.036,E2 -22361.036} C_VEL
LIN {X 0,Y 186.8,Z 440.411,A -85,B 0,C 180,E1 -22365.63,E2 -22365.63} C_VEL
LIN {X 0,Y 187.147,Z 442.395,A -85,B 0,C 180,E1 -22368.494,E2 -22368.494} C_VEL
LIN {X 0,Y 188.211,Z 445.466,A -85,B 0,C 180,E1 -22368.995,E2 -22368.995} C_VEL
LIN {X 0,Y 189.691,Z 447.934,A -85,B 0,C 180,E1 -22369.567,E2 -22369.567} C_VEL
LIN {X 0,Y 193.521,Z 457.357,A -85,B 0,C 180,E1 -22371.393,E2 -22371.393} C_VEL
LIN {X 0,Y 196.465,Z 469.633,A -85,B 0,C 180,E1 -22373.585,E2 -22373.585} C_VEL
LIN {X 0,Y 197.958,Z 481.196,A -85,B 0,C 180,E1 -22375.75,E2 -22375.75} C_VEL
LIN {X 0,Y 198.561,Z 492.602,A -85,B 0,C 180,E1 -22378.154,E2 -22378.154} C_VEL
LIN {X 0,Y 198.166,Z 502.581,A -85,B 0,C 180,E1 -22380.522,E2 -22380.522} C_VEL
LIN {X 0,Y 197.722,Z 505.779,A -85,B 0,C 180,E1 -22381.324,E2 -22381.324} C_VEL
LIN {X 0,Y 194.56,Z 514.929,A -85,B 0,C 180,E1 -22383.736,E2 -22383.736} C_VEL
LIN {X 0,Y 191.517,Z 523.82,A -85,B 0,C 180,E1 -22386.749,E2 -22386.749} C_VEL
LIN {X 0,Y 188.75,Z 531.04,A -85,B 0,C 180,E1 -22389.853,E2 -22389.853} C_VEL
LIN {X 0,Y 186.861,Z 535.89,A -85,B 0,C 180,E1 -22392.489,E2 -22392.489} C_VEL
LIN {X 0,Y 185.123,Z 540.608,A -85,B 0,C 180,E1 -22395.714,E2 -22395.714} C_VEL
LIN {X 0,Y 183.876,Z 544.588,A -85,B 0,C 180,E1 -22399.425,E2 -22399.425} C_VEL
LIN {X 0,Y 183.509,Z 546.081,A -85,B 0,C 180,E1 -22401.188,E2 -22401.188} C_VEL
LIN {X 0,Y 183.212,Z 547.479,A -85,B 0,C 180,E1 -22403.392,E2 -22403.392} C_VEL
LIN {X 0,Y 183.053,Z 549.09,A -85,B 0,C 180,E1 -22407.799,E2 -22407.799} C_VEL
LIN {X 0,Y 183.077,Z 549.194,A -85,B 0,C 180,E1 -22408.864,E2 -22408.864} C_VEL
LIN {X 0,Y 182.454,Z 549.253,A -85,B 0,C 180,E1 -22410.698,E2 -22410.698} C_VEL
LIN {X 0,Y 180.863,Z 548.979,A -85,B 0,C 180,E1 -22412.5,E2 -22412.5} C_VEL
LIN {X 0,Y 177.205,Z 547.625,A -85,B 0,C 180,E1 -22416.139,E2 -22416.139} C_VEL
LIN {X 0,Y 176.352,Z 546.572,A -85,B 0,C 180,E1 -22418.031,E2 -22418.031} C_VEL
LIN {X 0,Y 176.372,Z 546.143,A -85,B 0,C 180,E1 -22418.668,E2 -22418.668} C_VEL
LIN {X 0,Y 177.356,Z 542.88,A -85,B 0,C 180,E1 -22422.588,E2 -22422.588} C_VEL
LIN {X 0,Y 178.717,Z 538.886,A -85,B 0,C 180,E1 -22425.978,E2 -22425.978} C_VEL
LIN {X 0,Y 181.288,Z 532.759,A -85,B 0,C 180,E1 -22429.829,E2 -22429.829} C_VEL
LIN {X 0,Y 184.141,Z 525.684,A -85,B 0,C 180,E1 -22433.215,E2 -22433.215} C_VEL
LIN {X 0,Y 187.013,Z 517.768,A -85,B 0,C 180,E1 -22436.204,E2 -22436.204} C_VEL
LIN {X 0,Y 190.106,Z 509.26,A -85,B 0,C 180,E1 -22438.724,E2 -22438.724} C_VEL
LIN {X 0,Y 191.377,Z 505.344,A -85,B 0,C 180,E1 -22439.72,E2 -22439.72} C_VEL
LIN {X 0,Y 192.056,Z 495.004,A -85,B 0,C 180,E1 -22442.363,E2 -22442.363} C_VEL
LIN {X 0,Y 191.867,Z 485.662,A -85,B 0,C 180,E1 -22444.496,E2 -22444.496} C_VEL
LIN {X 0,Y 190.856,Z 474.565,A -85,B 0,C 180,E1 -22446.772,E2 -22446.772} C_VEL
LIN {X 0,Y 188.682,Z 463.242,A -85,B 0,C 180,E1 -22448.963,E2 -22448.963} C_VEL
LIN {X 0,Y 185.974,Z 455.019,A -85,B 0,C 180,E1 -22450.637,E2 -22450.637} C_VEL
LIN {X 0,Y 183.775,Z 450.339,A -85,B 0,C 180,E1 -22451.692,E2 -22451.692} C_VEL
LIN {X 0,Y 182.145,Z 446.824,A -85,B 0,C 180,E1 -22452.459,E2 -22452.459} C_VEL
LIN {X 0,Y 180.326,Z 443.686,A -85,B 0,C 180,E1 -22453.245,E2 -22453.245} C_VEL
LIN {X 0,Y 179.88,Z 442.053,A -85,B 0,C 180,E1 -22453.553,E2 -22453.553} C_VEL
LIN {X 0,Y 179.407,Z 439.121,A -85,B 0,C 180,E1 -22458.245,E2 -22458.245} C_VEL
LIN {X 0,Y 179.107,Z 437.108,A -85,B 0,C 180,E1 -22461.7,E2 -22461.7} C_VEL
LIN {X 0,Y 178.77,Z 434.474,A -85,B 0,C 180,E1 -22466.607,E2 -22466.607} C_VEL
LIN {X 0,Y 178.491,Z 433.254,A -85,B 0,C 180,E1 -22469.212,E2 -22469.212} C_VEL
LIN {X 0,Y 178.535,Z 433.247,A -85,B 0,C 180,E1 -22474.876,E2 -22474.876} C_VEL
LIN {X 0,Y 178.624,Z 433.236,A -85,B 0,C 180,E1 -22480.784,E2 -22480.784} C_VEL
LIN {X 0,Y 178.667,Z 433.23,A -85,B 0,C 180,E1 -22484.017,E2 -22484.017} C_VEL
LIN {X 0,Y 178.896,Z 433.201,A -85,B 0,C 180,E1 -22489.153,E2 -22489.153} C_VEL
LIN {X 0,Y 178.935,Z 433.191,A -85,B 0,C 180,E1 -22493.233,E2 -22493.233} C_VEL
LIN {X 0,Y 179.156,Z 433.167,A -85,B 0,C 180,E1 -22497.752,E2 -22497.752} C_VEL
LIN {X 0,Y 179.374,Z 433.141,A -85,B 0,C 180,E1 -22500,E2 -22500} C_VEL
LIN {X 0,Y 178.877,Z 433.203,A -85,B 0,C 180,E1 -22504.507,E2 -22504.507} C_VEL
LIN {X 0,Y 178.98,Z 433.19,A -85,B 0,C 180,E1 -22509.037,E2 -22509.037} C_VEL
LIN {X 0,Y 178.689,Z 433.225,A -85,B 0,C 180,E1 -22513.65,E2 -22513.65} C_VEL
LIN {X 0,Y 178.651,Z 433.228,A -85,B 0,C 180,E1 -22518.344,E2 -22518.344} C_VEL
LIN {X 0,Y 178.513,Z 433.247,A -85,B 0,C 180,E1 -22523.185,E2 -22523.185} C_VEL
LIN {X 0,Y 178.489,Z 433.251,A -85,B 0,C 180,E1 -22528.197,E2 -22528.197} C_VEL
LIN {X 0,Y 178.48,Z 433.251,A -85,B 0,C 180,E1 -22530.791,E2 -22530.791} C_VEL
LIN {X 0,Y 178.497,Z 433.249,A -85,B 0,C 180,E1 -22534.225,E2 -22534.225} C_VEL
LIN {X 0,Y 178.42,Z 433.26,A -85,B 0,C 180,E1 -22539.068,E2 -22539.068} C_VEL
LIN {X 0,Y 178.405,Z 433.263,A -85,B 0,C 180,E1 -22542.043,E2 -22542.043} C_VEL
LIN {X 0,Y 178.695,Z 435.105,A -85,B 0,C 180,E1 -22546.226,E2 -22546.226} C_VEL
LIN {X 0,Y 179.841,Z 438.026,A -85,B 0,C 180,E1 -22546.813,E2 -22546.813} C_VEL
LIN {X 0,Y 181.587,Z 440.666,A -85,B 0,C 180,E1 -22547.554,E2 -22547.554} C_VEL
LIN {X 0,Y 185.746,Z 448.867,A -85,B 0,C 180,E1 -22549.578,E2 -22549.578} C_VEL
LIN {X 0,Y 189.46,Z 458.737,A -85,B 0,C 180,E1 -22551.825,E2 -22551.825} C_VEL
LIN {X 0,Y 192.068,Z 469.272,A -85,B 0,C 180,E1 -22554.165,E2 -22554.165} C_VEL
LIN {X 0,Y 193.483,Z 478.252,A -85,B 0,C 180,E1 -22556.245,E2 -22556.245} C_VEL
LIN {X 0,Y 194.094,Z 489.188,A -85,B 0,C 180,E1 -22558.976,E2 -22558.976} C_VEL
LIN {X 0,Y 194.043,Z 491.339,A -85,B 0,C 180,E1 -22559.532,E2 -22559.532} C_VEL
LIN {X 0,Y 190.949,Z 500.985,A -85,B 0,C 180,E1 -22561.91,E2 -22561.91} C_VEL
LIN {X 0,Y 187.921,Z 509.443,A -85,B 0,C 180,E1 -22564.527,E2 -22564.527} C_VEL
LIN {X 0,Y 184.719,Z 517.433,A -85,B 0,C 180,E1 -22567.637,E2 -22567.637} C_VEL
LIN {X 0,Y 182.004,Z 523.841,A -85,B 0,C 180,E1 -22570.839,E2 -22570.839} C_VEL
LIN {X 0,Y 179.867,Z 528.92,A -85,B 0,C 180,E1 -22574.127,E2 -22574.127} C_VEL
LIN {X 0,Y 178.192,Z 532.864,A -85,B 0,C 180,E1 -22577.472,E2 -22577.472} C_VEL
LIN {X 0,Y 177.095,Z 535.771,A -85,B 0,C 180,E1 -22580.866,E2 -22580.866} C_VEL
LIN {X 0,Y 176.357,Z 538.018,A -85,B 0,C 180,E1 -22585.055,E2 -22585.055} C_VEL
LIN {X 0,Y 176.144,Z 538.753,A -85,B 0,C 180,E1 -22587.714,E2 -22587.714} C_VEL
LIN {X 0,Y 176.121,Z 538.979,A -85,B 0,C 180,E1 -22590,E2 -22590} C_VEL
LIN {X 0,Y 176.144,Z 538.784,A -85,B 0,C 180,E1 -22592.287,E2 -22592.287} C_VEL
LIN {X 0,Y 176.364,Z 538.06,A -85,B 0,C 180,E1 -22594.97,E2 -22594.97} C_VEL
LIN {X 0,Y 177.095,Z 535.875,A -85,B 0,C 180,E1 -22599.134,E2 -22599.134} C_VEL
LIN {X 0,Y 178.188,Z 533.007,A -85,B 0,C 180,E1 -22602.529,E2 -22602.529} C_VEL
LIN {X 0,Y 179.801,Z 529.115,A -85,B 0,C 180,E1 -22605.88,E2 -22605.88} C_VEL
LIN {X 0,Y 181.908,Z 524.093,A -85,B 0,C 180,E1 -22609.172,E2 -22609.172} C_VEL
LIN {X 0,Y 184.656,Z 517.76,A -85,B 0,C 180,E1 -22612.371,E2 -22612.371} C_VEL
LIN {X 0,Y 187.831,Z 509.84,A -85,B 0,C 180,E1 -22615.486,E2 -22615.486} C_VEL
LIN {X 0,Y 190.869,Z 501.133,A -85,B 0,C 180,E1 -22618.215,E2 -22618.215} C_VEL
LIN {X 0,Y 194.217,Z 490.854,A -85,B 0,C 180,E1 -22620.729,E2 -22620.729} C_VEL
LIN {X 0,Y 193.726,Z 480.165,A -85,B 0,C 180,E1 -22623.447,E2 -22623.447} C_VEL
LIN {X 0,Y 192.637,Z 471.981,A -85,B 0,C 180,E1 -22625.381,E2 -22625.381} C_VEL
LIN {X 0,Y 190.13,Z 460.843,A -85,B 0,C 180,E1 -22627.873,E2 -22627.873} C_VEL
LIN {X 0,Y 186.519,Z 450.633,A -85,B 0,C 180,E1 -22630.193,E2 -22630.193} C_VEL
LIN {X 0,Y 183.136,Z 443.634,A -85,B 0,C 180,E1 -22631.895,E2 -22631.895} C_VEL
LIN {X 0,Y 180.692,Z 439.212,A -85,B 0,C 180,E1 -22633.023,E2 -22633.023} C_VEL
LIN {X 0,Y 179.082,Z 436.404,A -85,B 0,C 180,E1 -22633.751,E2 -22633.751} C_VEL
LIN {X 0,Y 178.736,Z 435.017,A -85,B 0,C 180,E1 -22634.042,E2 -22634.042} C_VEL
LIN {X 0,Y 178.418,Z 433.262,A -85,B 0,C 180,E1 -22638.454,E2 -22638.454} C_VEL
LIN {X 0,Y 178.466,Z 433.253,A -85,B 0,C 180,E1 -22641.962,E2 -22641.962} C_VEL
LIN {X 0,Y 178.492,Z 433.248,A -85,B 0,C 180,E1 -22646.548,E2 -22646.548} C_VEL
LIN {X 0,Y 178.524,Z 433.243,A -85,B 0,C 180,E1 -22650.007,E2 -22650.007} C_VEL
LIN {X 0,Y 178.537,Z 433.241,A -85,B 0,C 180,E1 -22654.876,E2 -22654.876} C_VEL
LIN {X 0,Y 178.626,Z 433.235,A -85,B 0,C 180,E1 -22660.784,E2 -22660.784} C_VEL
LIN {X 0,Y 178.668,Z 433.231,A -85,B 0,C 180,E1 -22664.017,E2 -22664.017} C_VEL
LIN {X 0,Y 178.897,Z 433.2,A -85,B 0,C 180,E1 -22669.153,E2 -22669.153} C_VEL
LIN {X 0,Y 178.937,Z 433.196,A -85,B 0,C 180,E1 -22673.233,E2 -22673.233} C_VEL
LIN {X 0,Y 179.157,Z 433.168,A -85,B 0,C 180,E1 -22677.752,E2 -22677.752} C_VEL
LIN {X 0,Y 179.373,Z 433.14,A -85,B 0,C 180,E1 -22680,E2 -22680} C_VEL
LIN {X 0,Y 178.879,Z 433.203,A -85,B 0,C 180,E1 -22684.507,E2 -22684.507} C_VEL
LIN {X 0,Y 178.981,Z 433.19,A -85,B 0,C 180,E1 -22689.037,E2 -22689.037} C_VEL
LIN {X 0,Y 178.691,Z 433.226,A -85,B 0,C 180,E1 -22693.649,E2 -22693.649} C_VEL
LIN {X 0,Y 178.673,Z 433.228,A -85,B 0,C 180,E1 -22698.341,E2 -22698.341} C_VEL
LIN {X 0,Y 178.516,Z 433.25,A -85,B 0,C 180,E1 -22703.184,E2 -22703.184} C_VEL
LIN {X 0,Y 178.487,Z 433.247,A -85,B 0,C 180,E1 -22708.197,E2 -22708.197} C_VEL
LIN {X 0,Y 178.498,Z 433.268,A -85,B 0,C 180,E1 -22710.787,E2 -22710.787} C_VEL
LIN {X 0,Y 178.795,Z 435.041,A -85,B 0,C 180,E1 -22714.364,E2 -22714.364} C_VEL
LIN {X 0,Y 179.156,Z 437.5,A -85,B 0,C 180,E1 -22718.877,E2 -22718.877} C_VEL
LIN {X 0,Y 179.443,Z 439.275,A -85,B 0,C 180,E1 -22721.914,E2 -22721.914} C_VEL
LIN {X 0,Y 179.924,Z 442.257,A -85,B 0,C 180,E1 -22726.433,E2 -22726.433} C_VEL
LIN {X 0,Y 181.006,Z 445.244,A -85,B 0,C 180,E1 -22726.984,E2 -22726.984} C_VEL
LIN {X 0,Y 182.64,Z 447.798,A -85,B 0,C 180,E1 -22727.664,E2 -22727.664} C_VEL
LIN {X 0,Y 186.475,Z 456.206,A -85,B 0,C 180,E1 -22729.539,E2 -22729.539} C_VEL
LIN {X 0,Y 188.251,Z 461.411,A -85,B 0,C 180,E1 -22730.604,E2 -22730.604} C_VEL
LIN {X 0,Y 190.637,Z 472.636,A -85,B 0,C 180,E1 -22732.782,E2 -22732.782} C_VEL
LIN {X 0,Y 191.894,Z 484.664,A -85,B 0,C 180,E1 -22735.235,E2 -22735.235} C_VEL
LIN {X 0,Y 192.134,Z 495.094,A -85,B 0,C 180,E1 -22737.601,E2 -22737.601} C_VEL
LIN {X 0,Y 191.434,Z 505.575,A -85,B 0,C 180,E1 -22740.289,E2 -22740.289} C_VEL
LIN {X 0,Y 188.183,Z 514.726,A -85,B 0,C 180,E1 -22742.774,E2 -22742.774} C_VEL
LIN {X 0,Y 185.198,Z 522.943,A -85,B 0,C 180,E1 -22745.612,E2 -22745.612} C_VEL
LIN {X 0,Y 182.515,Z 529.721,A -85,B 0,C 180,E1 -22748.542,E2 -22748.542} C_VEL
LIN {X 0,Y 180.082,Z 535.687,A -85,B 0,C 180,E1 -22751.807,E2 -22751.807} C_VEL
LIN {X 0,Y 178.197,Z 540.404,A -85,B 0,C 180,E1 -22755.146,E2 -22755.146} C_VEL
LIN {X 0,Y 177,Z 544.014,A -85,B 0,C 180,E1 -22758.549,E2 -22758.549} C_VEL
LIN {X 0,Y 176.468,Z 545.876,A -85,B 0,C 180,E1 -22760.833,E2 -22760.833} C_VEL
LIN {X 0,Y 176.14,Z 547.275,A -85,B 0,C 180,E1 -22763.125,E2 -22763.125} C_VEL
LIN {X 0,Y 175.969,Z 548.886,A -85,B 0,C 180,E1 -22767.711,E2 -22767.711} C_VEL
LIN {X 0,Y 176.079,Z 549.102,A -85,B 0,C 180,E1 -22770,E2 -22770} C_VEL
LIN {X 0,Y 175.947,Z 548.714,A -85,B 0,C 180,E1 -22773.034,E2 -22773.034} C_VEL
LIN {X 0,Y 176.139,Z 547.247,A -85,B 0,C 180,E1 -22776.875,E2 -22776.875} C_VEL
LIN {X 0,Y 176.372,Z 546.143,A -85,B 0,C 180,E1 -22778.668,E2 -22778.668} C_VEL
LIN {X 0,Y 176.096,Z 544.834,A -85,B 0,C 180,E1 -22780.538,E2 -22780.538} C_VEL
LIN {X 0,Y 174.138,Z 542.084,A -85,B 0,C 180,E1 -22783.591,E2 -22783.591} C_VEL
LIN {X 0,Y 172.602,Z 538.621,A -85,B 0,C 180,E1 -22786.626,E2 -22786.626} C_VEL
LIN {X 0,Y 172.987,Z 536.152,A -85,B 0,C 180,E1 -22788.408,E2 -22788.408} C_VEL
LIN {X 0,Y 175.419,Z 530.508,A -85,B 0,C 180,E1 -22791.752,E2 -22791.752} C_VEL
LIN {X 0,Y 178.559,Z 523.057,A -85,B 0,C 180,E1 -22795.14,E2 -22795.14} C_VEL
LIN {X 0,Y 181.88,Z 514.333,A -85,B 0,C 180,E1 -22798.252,E2 -22798.252} C_VEL
LIN {X 0,Y 184.579,Z 507.099,A -85,B 0,C 180,E1 -22800.298,E2 -22800.298} C_VEL
LIN {X 0,Y 185.581,Z 498.417,A -85,B 0,C 180,E1 -22802.676,E2 -22802.676} C_VEL
LIN {X 0,Y 185.677,Z 489.01,A -85,B 0,C 180,E1 -22805.016,E2 -22805.016} C_VEL
LIN {X 0,Y 185.032,Z 478.209,A -85,B 0,C 180,E1 -22807.425,E2 -22807.425} C_VEL
LIN {X 0,Y 183.545,Z 468.413,A -85,B 0,C 180,E1 -22809.48,E2 -22809.48} C_VEL
LIN {X 0,Y 181.38,Z 460.484,A -85,B 0,C 180,E1 -22811.201,E2 -22811.201} C_VEL
LIN {X 0,Y 178.508,Z 453.736,A -85,B 0,C 180,E1 -22812.838,E2 -22812.838} C_VEL
LIN {X 0,Y 177.069,Z 450.862,A -85,B 0,C 180,E1 -22813.57,E2 -22813.57} C_VEL
LIN {X 0,Y 174.932,Z 446.623,A -85,B 0,C 180,E1 -22814.651,E2 -22814.651} C_VEL
LIN {X 0,Y 173.063,Z 443.344,A -85,B 0,C 180,E1 -22815.554,E2 -22815.554} C_VEL
LIN {X 0,Y 172.612,Z 441.77,A -85,B 0,C 180,E1 -22815.912,E2 -22815.912} C_VEL
LIN {X 0,Y 172.182,Z 438.921,A -85,B 0,C 180,E1 -22820.853,E2 -22820.853} C_VEL
LIN {X 0,Y 171.898,Z 436.678,A -85,B 0,C 180,E1 -22825.083,E2 -22825.083} C_VEL
LIN {X 0,Y 171.451,Z 434.13,A -85,B 0,C 180,E1 -22830.535,E2 -22830.535} C_VEL
LIN {X 0,Y 171.459,Z 434.128,A -85,B 0,C 180,E1 -22835.802,E2 -22835.802} C_VEL
LIN {X 0,Y 171.58,Z 434.114,A -85,B 0,C 180,E1 -22840.872,E2 -22840.872} C_VEL
LIN {X 0,Y 171.611,Z 434.109,A -85,B 0,C 180,E1 -22845.776,E2 -22845.776} C_VEL
LIN {X 0,Y 171.912,Z 434.07,A -85,B 0,C 180,E1 -22850.588,E2 -22850.588} C_VEL
LIN {X 0,Y 171.827,Z 434.08,A -85,B 0,C 180,E1 -22855.308,E2 -22855.308} C_VEL
LIN {X 0,Y 172.337,Z 434.017,A -85,B 0,C 180,E1 -22860,E2 -22860} C_VEL
LIN {X 0,Y 171.827,Z 434.081,A -85,B 0,C 180,E1 -22864.692,E2 -22864.692} C_VEL
LIN {X 0,Y 171.912,Z 434.071,A -85,B 0,C 180,E1 -22869.412,E2 -22869.412} C_VEL
LIN {X 0,Y 171.611,Z 434.109,A -85,B 0,C 180,E1 -22874.224,E2 -22874.224} C_VEL
LIN {X 0,Y 171.546,Z 434.109,A -85,B 0,C 180,E1 -22879.562,E2 -22879.562} C_VEL
LIN {X 0,Y 171.47,Z 434.126,A -85,B 0,C 180,E1 -22885.617,E2 -22885.617} C_VEL
LIN {X 0,Y 171.443,Z 434.128,A -85,B 0,C 180,E1 -22890.587,E2 -22890.587} C_VEL
LIN {X 0,Y 171.408,Z 434.133,A -85,B 0,C 180,E1 -22895.032,E2 -22895.032} C_VEL
LIN {X 0,Y 171.381,Z 434.137,A -85,B 0,C 180,E1 -22898.817,E2 -22898.817} C_VEL
LIN {X 0,Y 171.346,Z 434.142,A -85,B 0,C 180,E1 -22901.016,E2 -22901.016} C_VEL
LIN {X 0,Y 171.542,Z 435.5,A -85,B 0,C 180,E1 -22903.896,E2 -22903.896} C_VEL
LIN {X 0,Y 172.693,Z 438.301,A -85,B 0,C 180,E1 -22904.541,E2 -22904.541} C_VEL
LIN {X 0,Y 174.627,Z 441.029,A -85,B 0,C 180,E1 -22905.435,E2 -22905.435} C_VEL
LIN {X 0,Y 179.322,Z 450.032,A -85,B 0,C 180,E1 -22907.92,E2 -22907.92} C_VEL
LIN {X 0,Y 182.924,Z 459.081,A -85,B 0,C 180,E1 -22910.212,E2 -22910.212} C_VEL
LIN {X 0,Y 185.32,Z 467.882,A -85,B 0,C 180,E1 -22912.323,E2 -22912.323} C_VEL
LIN {X 0,Y 187.048,Z 478.123,A -85,B 0,C 180,E1 -22914.834,E2 -22914.834} C_VEL
LIN {X 0,Y 187.647,Z 487.72,A -85,B 0,C 180,E1 -22917.32,E2 -22917.32} C_VEL
LIN {X 0,Y 187.604,Z 492.618,A -85,B 0,C 180,E1 -22918.682,E2 -22918.682} C_VEL
LIN {X 0,Y 184.612,Z 501.501,A -85,B 0,C 180,E1 -22920.963,E2 -22920.963} C_VEL
LIN {X 0,Y 180.984,Z 511.128,A -85,B 0,C 180,E1 -22924.096,E2 -22924.096} C_VEL
LIN {X 0,Y 177.665,Z 518.804,A -85,B 0,C 180,E1 -22927.314,E2 -22927.314} C_VEL
LIN {X 0,Y 174.492,Z 525.852,A -85,B 0,C 180,E1 -22931.203,E2 -22931.203} C_VEL
LIN {X 0,Y 172.373,Z 530.542,A -85,B 0,C 180,E1 -22934.632,E2 -22934.632} C_VEL
LIN {X 0,Y 170.819,Z 534.127,A -85,B 0,C 180,E1 -22938.129,E2 -22938.129} C_VEL
LIN {X 0,Y 170.099,Z 535.976,A -85,B 0,C 180,E1 -22940.487,E2 -22940.487} C_VEL
LIN {X 0,Y 169.585,Z 537.364,A -85,B 0,C 180,E1 -22942.858,E2 -22942.858} C_VEL
LIN {X 0,Y 169.258,Z 538.35,A -85,B 0,C 180,E1 -22945.237,E2 -22945.237} C_VEL
LIN {X 0,Y 169.063,Z 538.957,A -85,B 0,C 180,E1 -22947.618,E2 -22947.618} C_VEL
LIN {X 0,Y 169.033,Z 539.183,A -85,B 0,C 180,E1 -22950,E2 -22950} C_VEL
LIN {X 0,Y 169.062,Z 538.988,A -85,B 0,C 180,E1 -22952.383,E2 -22952.383} C_VEL
LIN {X 0,Y 169.258,Z 538.402,A -85,B 0,C 180,E1 -22954.764,E2 -22954.764} C_VEL
LIN {X 0,Y 170.099,Z 536.078,A -85,B 0,C 180,E1 -22959.513,E2 -22959.513} C_VEL
LIN {X 0,Y 171.268,Z 533.21,A -85,B 0,C 180,E1 -22963.044,E2 -22963.044} C_VEL
LIN {X 0,Y 172.974,Z 529.318,A -85,B 0,C 180,E1 -22966.524,E2 -22966.524} C_VEL
LIN {X 0,Y 175.212,Z 524.295,A -85,B 0,C 180,E1 -22969.935,E2 -22969.935} C_VEL
LIN {X 0,Y 178.112,Z 517.962,A -85,B 0,C 180,E1 -22973.24,E2 -22973.24} C_VEL
LIN {X 0,Y 181.434,Z 510.042,A -85,B 0,C 180,E1 -22976.453,E2 -22976.453} C_VEL
LIN {X 0,Y 184.577,Z 501.482,A -85,B 0,C 180,E1 -22979.216,E2 -22979.216} C_VEL
LIN {X 0,Y 187.794,Z 492.116,A -85,B 0,C 180,E1 -22981.597,E2 -22981.597} C_VEL
LIN {X 0,Y 187.536,Z 482.519,A -85,B 0,C 180,E1 -22984.204,E2 -22984.204} C_VEL
LIN {X 0,Y 186.298,Z 472.523,A -85,B 0,C 180,E1 -22986.714,E2 -22986.714} C_VEL
LIN {X 0,Y 183.902,Z 462.039,A -85,B 0,C 180,E1 -22989.244,E2 -22989.244} C_VEL
LIN {X 0,Y 180.392,Z 452.195,A -85,B 0,C 180,E1 -22991.688,E2 -22991.688} C_VEL
LIN {X 0,Y 176.113,Z 443.87,A -85,B 0,C 180,E1 -22993.982,E2 -22993.982} C_VEL
LIN {X 0,Y 173.992,Z 439.942,A -85,B 0,C 180,E1 -22995.075,E2 -22995.075} C_VEL
LIN {X 0,Y 172.029,Z 437.024,A -85,B 0,C 180,E1 -22996.011,E2 -22996.011} C_VEL
LIN {X 0,Y 171.505,Z 435.33,A -85,B 0,C 180,E1 -22996.34,E2 -22996.34} C_VEL
LIN {X 0,Y 171.354,Z 434.209,A -85,B 0,C 180,E1 -22998.987,E2 -22998.987} C_VEL
LIN {X 0,Y 171.416,Z 434.131,A -85,B 0,C 180,E1 -23002.048,E2 -23002.048} C_VEL
LIN {X 0,Y 171.412,Z 434.133,A -85,B 0,C 180,E1 -23005.087,E2 -23005.087} C_VEL
LIN {X 0,Y 171.45,Z 434.124,A -85,B 0,C 180,E1 -23010.534,E2 -23010.534} C_VEL
LIN {X 0,Y 171.46,Z 434.126,A -85,B 0,C 180,E1 -23015.802,E2 -23015.802} C_VEL
LIN {X 0,Y 171.582,Z 434.112,A -85,B 0,C 180,E1 -23020.872,E2 -23020.872} C_VEL
LIN {X 0,Y 171.612,Z 434.106,A -85,B 0,C 180,E1 -23025.776,E2 -23025.776} C_VEL
LIN {X 0,Y 171.913,Z 434.068,A -85,B 0,C 180,E1 -23030.588,E2 -23030.588} C_VEL
LIN {X 0,Y 171.828,Z 434.081,A -85,B 0,C 180,E1 -23035.308,E2 -23035.308} C_VEL
LIN {X 0,Y 172.336,Z 434.017,A -85,B 0,C 180,E1 -23040,E2 -23040} C_VEL
LIN {X 0,Y 171.828,Z 434.081,A -85,B 0,C 180,E1 -23044.692,E2 -23044.692} C_VEL
LIN {X 0,Y 171.913,Z 434.072,A -85,B 0,C 180,E1 -23049.411,E2 -23049.411} C_VEL
LIN {X 0,Y 171.616,Z 434.108,A -85,B 0,C 180,E1 -23054.224,E2 -23054.224} C_VEL
LIN {X 0,Y 171.56,Z 434.115,A -85,B 0,C 180,E1 -23059.574,E2 -23059.574} C_VEL
LIN {X 0,Y 171.471,Z 434.126,A -85,B 0,C 180,E1 -23065.616,E2 -23065.616} C_VEL
LIN {X 0,Y 171.457,Z 434.181,A -85,B 0,C 180,E1 -23069.464,E2 -23069.464} C_VEL
LIN {X 0,Y 171.859,Z 436.756,A -85,B 0,C 180,E1 -23074.926,E2 -23074.926} C_VEL
LIN {X 0,Y 172.184,Z 438.984,A -85,B 0,C 180,E1 -23079.147,E2 -23079.147} C_VEL
LIN {X 0,Y 172.643,Z 441.859,A -85,B 0,C 180,E1 -23084.08,E2 -23084.08} C_VEL
LIN {X 0,Y 173.698,Z 444.81,A -85,B 0,C 180,E1 -23084.677,E2 -23084.677} C_VEL
LIN {X 0,Y 175.6,Z 447.75,A -85,B 0,C 180,E1 -23085.553,E2 -23085.553} C_VEL
LIN {X 0,Y 177.534,Z 451.581,A -85,B 0,C 180,E1 -23086.543,E2 -23086.543} C_VEL
LIN {X 0,Y 181.013,Z 459.309,A -85,B 0,C 180,E1 -23088.449,E2 -23088.449} C_VEL
LIN {X 0,Y 182.891,Z 465.242,A -85,B 0,C 180,E1 -23089.768,E2 -23089.768} C_VEL
LIN {X 0,Y 184.892,Z 476.315,A -85,B 0,C 180,E1 -23092.093,E2 -23092.093} C_VEL
LIN {X 0,Y 185.737,Z 487.42,A -85,B 0,C 180,E1 -23094.552,E2 -23094.552} C_VEL
LIN {X 0,Y 185.71,Z 497.246,A -85,B 0,C 180,E1 -23096.954,E2 -23096.954} C_VEL
LIN {X 0,Y 185.041,Z 505.365,A -85,B 0,C 180,E1 -23099.153,E2 -23099.153} C_VEL
LIN {X 0,Y 183.911,Z 509.274,A -85,B 0,C 180,E1 -23100.212,E2 -23100.212} C_VEL
LIN {X 0,Y 180.655,Z 517.735,A -85,B 0,C 180,E1 -23102.799,E2 -23102.799} C_VEL
LIN {X 0,Y 177.474,Z 525.925,A -85,B 0,C 180,E1 -23106.012,E2 -23106.012} C_VEL
LIN {X 0,Y 174.574,Z 532.669,A -85,B 0,C 180,E1 -23109.374,E2 -23109.374} C_VEL
LIN {X 0,Y 171.879,Z 538.764,A -85,B 0,C 180,E1 -23113.368,E2 -23113.368} C_VEL
LIN {X 0,Y 170.408,Z 542.735,A -85,B 0,C 180,E1 -23116.889,E2 -23116.889} C_VEL
LIN {X 0,Y 169.425,Z 545.672,A -85,B 0,C 180,E1 -23120.449,E2 -23120.449} C_VEL
LIN {X 0,Y 169.074,Z 547.071,A -85,B 0,C 180,E1 -23122.836,E2 -23122.836} C_VEL
LIN {X 0,Y 168.863,Z 548.682,A -85,B 0,C 180,E1 -23127.614,E2 -23127.614} C_VEL
LIN {X 0,Y 168.988,Z 548.898,A -85,B 0,C 180,E1 -23130,E2 -23130} C_VEL
LIN {X 0,Y 168.857,Z 548.609,A -85,B 0,C 180,E1 -23132.678,E2 -23132.678} C_VEL
LIN {X 0,Y 169.074,Z 547.042,A -85,B 0,C 180,E1 -23137.163,E2 -23137.163} C_VEL
LIN {X 0,Y 169.425,Z 545.63,A -85,B 0,C 180,E1 -23139.551,E2 -23139.551} C_VEL
LIN {X 0,Y 170.407,Z 542.674,A -85,B 0,C 180,E1 -23143.11,E2 -23143.11} C_VEL
LIN {X 0,Y 171.878,Z 538.68,A -85,B 0,C 180,E1 -23146.632,E2 -23146.632} C_VEL
LIN {X 0,Y 172.987,Z 536.152,A -85,B 0,C 180,E1 -23148.408,E2 -23148.408} C_VEL
LIN {X 0,Y 173.527,Z 533.514,A -85,B 0,C 180,E1 -23150.151,E2 -23150.151} C_VEL
LIN {X 0,Y 172.888,Z 528.831,A -85,B 0,C 180,E1 -23153.043,E2 -23153.043} C_VEL
LIN {X 0,Y 172.477,Z 523.505,A -85,B 0,C 180,E1 -23155.826,E2 -23155.826} C_VEL
LIN {X 0,Y 173.339,Z 519.858,A -85,B 0,C 180,E1 -23157.348,E2 -23157.348} C_VEL
LIN {X 0,Y 177.027,Z 510.65,A -85,B 0,C 180,E1 -23160.409,E2 -23160.409} C_VEL
LIN {X 0,Y 178.33,Z 506.887,A -85,B 0,C 180,E1 -23161.479,E2 -23161.479} C_VEL
LIN {X 0,Y 179.269,Z 498.055,A -85,B 0,C 180,E1 -23164.02,E2 -23164.02} C_VEL
LIN {X 0,Y 179.415,Z 489.1,A -85,B 0,C 180,E1 -23166.353,E2 -23166.353} C_VEL
LIN {X 0,Y 178.807,Z 477.976,A -85,B 0,C 180,E1 -23168.967,E2 -23168.967} C_VEL
LIN {X 0,Y 177.274,Z 468.43,A -85,B 0,C 180,E1 -23171.127,E2 -23171.127} C_VEL
LIN {X 0,Y 174.957,Z 461.103,A -85,B 0,C 180,E1 -23172.938,E2 -23172.938} C_VEL
LIN {X 0,Y 171.975,Z 454.529,A -85,B 0,C 180,E1 -23174.761,E2 -23174.761} C_VEL
LIN {X 0,Y 170.304,Z 451.169,A -85,B 0,C 180,E1 -23175.708,E2 -23175.708} C_VEL
LIN {X 0,Y 168.436,Z 447.264,A -85,B 0,C 180,E1 -23176.788,E2 -23176.788} C_VEL
LIN {X 0,Y 166.106,Z 443.84,A -85,B 0,C 180,E1 -23177.977,E2 -23177.977} C_VEL
LIN {X 0,Y 165.379,Z 441.501,A -85,B 0,C 180,E1 -23178.527,E2 -23178.527} C_VEL
LIN {X 0,Y 164.977,Z 438.594,A -85,B 0,C 180,E1 -23184.037,E2 -23184.037} C_VEL
LIN {X 0,Y 164.623,Z 436.205,A -85,B 0,C 180,E1 -23189.183,E2 -23189.183} C_VEL
LIN {X 0,Y 164.364,Z 435.057,A -85,B 0,C 180,E1 -23191.943,E2 -23191.943} C_VEL
LIN {X 0,Y 164.417,Z 435.006,A -85,B 0,C 180,E1 -23194.694,E2 -23194.694} C_VEL
LIN {X 0,Y 164.485,Z 434.997,A -85,B 0,C 180,E1 -23200.051,E2 -23200.051} C_VEL
LIN {X 0,Y 164.555,Z 434.989,A -85,B 0,C 180,E1 -23205.152,E2 -23205.152} C_VEL
LIN {X 0,Y 164.854,Z 434.95,A -85,B 0,C 180,E1 -23210.182,E2 -23210.182} C_VEL
LIN {X 0,Y 164.863,Z 434.946,A -85,B 0,C 180,E1 -23212.653,E2 -23212.653} C_VEL
LIN {X 0,Y 165.299,Z 434.894,A -85,B 0,C 180,E1 -23220,E2 -23220} C_VEL
LIN {X 0,Y 164.863,Z 434.949,A -85,B 0,C 180,E1 -23227.348,E2 -23227.348} C_VEL
LIN {X 0,Y 164.781,Z 434.957,A -85,B 0,C 180,E1 -23231.198,E2 -23231.198} C_VEL
LIN {X 0,Y 164.508,Z 434.994,A -85,B 0,C 180,E1 -23237.401,E2 -23237.401} C_VEL
LIN {X 0,Y 164.474,Z 434.99,A -85,B 0,C 180,E1 -23239.989,E2 -23239.989} C_VEL
LIN {X 0,Y 164.395,Z 435.007,A -85,B 0,C 180,E1 -23246.134,E2 -23246.134} C_VEL
LIN {X 0,Y 164.377,Z 435.008,A -85,B 0,C 180,E1 -23251.229,E2 -23251.229} C_VEL
LIN {X 0,Y 164.314,Z 435.018,A -85,B 0,C 180,E1 -23256.785,E2 -23256.785} C_VEL
LIN {X 0,Y 164.301,Z 435.102,A -85,B 0,C 180,E1 -23259.914,E2 -23259.914} C_VEL
LIN {X 0,Y 164.409,Z 435.588,A -85,B 0,C 180,E1 -23261.191,E2 -23261.191} C_VEL
LIN {X 0,Y 165.551,Z 438.534,A -85,B 0,C 180,E1 -23261.961,E2 -23261.961} C_VEL
LIN {X 0,Y 167.572,Z 441.262,A -85,B 0,C 180,E1 -23262.999,E2 -23262.999} C_VEL
LIN {X 0,Y 169.685,Z 445.017,A -85,B 0,C 180,E1 -23264.2,E2 -23264.2} C_VEL
LIN {X 0,Y 173.879,Z 453.166,A -85,B 0,C 180,E1 -23266.681,E2 -23266.681} C_VEL
LIN {X 0,Y 176.837,Z 460.663,A -85,B 0,C 180,E1 -23268.776,E2 -23268.776} C_VEL
LIN {X 0,Y 179.084,Z 468.779,A -85,B 0,C 180,E1 -23270.902,E2 -23270.902} C_VEL
LIN {X 0,Y 180.825,Z 479.235,A -85,B 0,C 180,E1 -23273.651,E2 -23273.651} C_VEL
LIN {X 0,Y 181.318,Z 488.448,A -85,B 0,C 180,E1 -23276.174,E2 -23276.174} C_VEL
LIN {X 0,Y 181.206,Z 493.891,A -85,B 0,C 180,E1 -23277.772,E2 -23277.772} C_VEL
LIN {X 0,Y 177.895,Z 503.123,A -85,B 0,C 180,E1 -23280.276,E2 -23280.276} C_VEL
LIN {X 0,Y 174.626,Z 511.334,A -85,B 0,C 180,E1 -23283.079,E2 -23283.079} C_VEL
LIN {X 0,Y 171.147,Z 519.01,A -85,B 0,C 180,E1 -23286.399,E2 -23286.399} C_VEL
LIN {X 0,Y 167.767,Z 526.059,A -85,B 0,C 180,E1 -23290.42,E2 -23290.42} C_VEL
LIN {X 0,Y 165.535,Z 530.747,A -85,B 0,C 180,E1 -23293.981,E2 -23293.981} C_VEL
LIN {X 0,Y 163.876,Z 534.332,A -85,B 0,C 180,E1 -23297.618,E2 -23297.618} C_VEL
LIN {X 0,Y 163.086,Z 536.181,A -85,B 0,C 180,E1 -23300.074,E2 -23300.074} C_VEL
LIN {X 0,Y 162.548,Z 537.568,A -85,B 0,C 180,E1 -23302.547,E2 -23302.547} C_VEL
LIN {X 0,Y 162.125,Z 538.733,A -85,B 0,C 180,E1 -23305.588,E2 -23305.588} C_VEL
LIN {X 0,Y 161.946,Z 539.386,A -85,B 0,C 180,E1 -23310,E2 -23310} C_VEL
LIN {X 0,Y 162.126,Z 538.784,A -85,B 0,C 180,E1 -23314.413,E2 -23314.413} C_VEL
LIN {X 0,Y 162.548,Z 537.638,A -85,B 0,C 180,E1 -23317.453,E2 -23317.453} C_VEL
LIN {X 0,Y 163.085,Z 536.282,A -85,B 0,C 180,E1 -23319.926,E2 -23319.926} C_VEL
LIN {X 0,Y 164.342,Z 533.414,A -85,B 0,C 180,E1 -23323.604,E2 -23323.604} C_VEL
LIN {X 0,Y 166.178,Z 529.521,A -85,B 0,C 180,E1 -23327.22,E2 -23327.22} C_VEL
LIN {X 0,Y 168.554,Z 524.498,A -85,B 0,C 180,E1 -23330.758,E2 -23330.758} C_VEL
LIN {X 0,Y 171.609,Z 518.164,A -85,B 0,C 180,E1 -23334.176,E2 -23334.176} C_VEL
LIN {X 0,Y 175.051,Z 510.353,A -85,B 0,C 180,E1 -23337.45,E2 -23337.45} C_VEL
LIN {X 0,Y 178.222,Z 502.174,A -85,B 0,C 180,E1 -23340.184,E2 -23340.184} C_VEL
LIN {X 0,Y 181.391,Z 493.383,A -85,B 0,C 180,E1 -23342.52,E2 -23342.52} C_VEL
LIN {X 0,Y 181.314,Z 484.567,A -85,B 0,C 180,E1 -23345.062,E2 -23345.062} C_VEL
LIN {X 0,Y 180.298,Z 475.025,A -85,B 0,C 180,E1 -23347.636,E2 -23347.636} C_VEL
LIN {X 0,Y 178.637,Z 466.506,A -85,B 0,C 180,E1 -23349.847,E2 -23349.847} C_VEL
LIN {X 0,Y 175.752,Z 457.418,A -85,B 0,C 180,E1 -23352.289,E2 -23352.289} C_VEL
LIN {X 0,Y 171.775,Z 448.903,A -85,B 0,C 180,E1 -23354.797,E2 -23354.797} C_VEL
LIN {X 0,Y 169.548,Z 444.795,A -85,B 0,C 180,E1 -23356.084,E2 -23356.084} C_VEL
LIN {X 0,Y 167.609,Z 441.283,A -85,B 0,C 180,E1 -23357.2,E2 -23357.2} C_VEL
LIN {X 0,Y 164.996,Z 437.511,A -85,B 0,C 180,E1 -23358.581,E2 -23358.581} C_VEL
LIN {X 0,Y 164.396,Z 435.61,A -85,B 0,C 180,E1 -23359.008,E2 -23359.008} C_VEL
LIN {X 0,Y 164.309,Z 435.098,A -85,B 0,C 180,E1 -23360.347,E2 -23360.347} C_VEL
LIN {X 0,Y 164.345,Z 435.011,A -85,B 0,C 180,E1 -23364.343,E2 -23364.343} C_VEL
LIN {X 0,Y 164.391,Z 435.007,A -85,B 0,C 180,E1 -23369.135,E2 -23369.135} C_VEL
LIN {X 0,Y 164.418,Z 434.998,A -85,B 0,C 180,E1 -23374.694,E2 -23374.694} C_VEL
LIN {X 0,Y 164.487,Z 434.995,A -85,B 0,C 180,E1 -23380.051,E2 -23380.051} C_VEL
LIN {X 0,Y 164.556,Z 434.985,A -85,B 0,C 180,E1 -23385.152,E2 -23385.152} C_VEL
LIN {X 0,Y 164.856,Z 434.949,A -85,B 0,C 180,E1 -23390.181,E2 -23390.181} C_VEL
LIN {X 0,Y 164.865,Z 434.949,A -85,B 0,C 180,E1 -23392.652,E2 -23392.652} C_VEL
LIN {X 0,Y 165.053,Z 434.924,A -85,B 0,C 180,E1 -23397.559,E2 -23397.559} C_VEL
LIN {X 0,Y 165.298,Z 434.893,A -85,B 0,C 180,E1 -23400,E2 -23400} C_VEL
LIN {X 0,Y 164.778,Z 434.959,A -85,B 0,C 180,E1 -23404.893,E2 -23404.893} C_VEL
LIN {X 0,Y 164.865,Z 434.949,A -85,B 0,C 180,E1 -23407.347,E2 -23407.347} C_VEL
LIN {X 0,Y 164.782,Z 434.957,A -85,B 0,C 180,E1 -23411.198,E2 -23411.198} C_VEL
LIN {X 0,Y 164.522,Z 434.991,A -85,B 0,C 180,E1 -23417.399,E2 -23417.399} C_VEL
LIN {X 0,Y 164.477,Z 434.996,A -85,B 0,C 180,E1 -23419.989,E2 -23419.989} C_VEL
LIN {X 0,Y 164.395,Z 435.006,A -85,B 0,C 180,E1 -23426.133,E2 -23426.133} C_VEL
LIN {X 0,Y 164.383,Z 435.118,A -85,B 0,C 180,E1 -23428.053,E2 -23428.053} C_VEL
LIN {X 0,Y 164.643,Z 436.525,A -85,B 0,C 180,E1 -23431.38,E2 -23431.38} C_VEL
LIN {X 0,Y 164.987,Z 438.987,A -85,B 0,C 180,E1 -23436.61,E2 -23436.61} C_VEL
LIN {X 0,Y 165.368,Z 441.514,A -85,B 0,C 180,E1 -23441.38,E2 -23441.38} C_VEL
LIN {X 0,Y 166.47,Z 444.545,A -85,B 0,C 180,E1 -23442.103,E2 -23442.103} C_VEL
LIN {X 0,Y 168.562,Z 447.645,A -85,B 0,C 180,E1 -23443.172,E2 -23443.172} C_VEL
